Yaskawa INFORM job: SKRZYNIA_4640_-90_STOPNI_10BR.JBI

/JOB
//NAME SKRZYNIA_4640_-90_STOPNI_10BR
///FOLDERNAME 02-SKRZYNIE_JOBS
//POS
///NPOS 666,666,0,47,0,0
///TOOL 0
///POSTYPE PULSE
///PULSE
C00000=0,-52280,40443,0,6876,0
C00001=-82314,-24956,17040,-59626,-27382,-6248
C00002=-93910,-8625,17040,-59626,-43355,-6248
C00003=-98846,-1061,-42166,-80308,-57081,16120
C00004=-100452,6057,-48127,-85711,-56704,21322
C00005=-96957,25597,-37888,-85158,-62082,25522
C00006=-95580,33075,-33256,-84644,-64024,26851
C00007=-94380,33739,-32188,-85134,-63496,26721
C00008=-95580,33075,-33256,-84644,-64024,26851
C00009=-94940,31262,-36138,-85248,-63712,27160
C00010=-95580,33075,-33256,-84644,-64024,26851
C00011=-95263,33142,-33256,-84677,-63995,26850
C00012=-95263,33142,-33256,-84677,-63995,26850
C00013=-94261,33702,-32359,-85087,-63552,26740
C00014=-95263,33142,-33256,-84677,-63995,26850
C00015=-94777,31773,-35433,-85135,-63758,27084
C00016=-95263,33142,-33256,-84677,-63995,26850
C00017=-95260,33144,-33256,-84678,-63995,26850
C00018=-95260,33144,-33256,-84678,-63995,26850
C00019=-94282,33689,-32380,-85076,-63563,26742
C00020=-95260,33144,-33256,-84678,-63995,26850
C00021=-94827,31920,-35204,-85086,-63784,27059
C00022=-95260,33144,-33256,-84678,-63995,26850
C00023=-95258,33145,-33257,-84676,-63996,26846
C00024=-95258,33145,-33257,-84676,-63996,26846
C00025=-94286,33686,-32387,-85074,-63568,26738
C00026=-95258,33145,-33257,-84676,-63996,26846
C00027=-94874,32057,-34990,-85039,-63809,27032
C00028=-95258,33145,-33257,-84676,-63996,26846
C00029=-95377,22848,-19980,-77610,-66139,18413
C00030=-95383,22536,-19091,-77284,-66299,17999
C00031=-94454,23123,-18267,-77513,-65785,17889
C00032=-95383,22536,-19091,-77284,-66299,17999
C00033=-94991,21279,-20843,-77511,-66022,18108
C00034=-95383,22536,-19091,-77284,-66299,17999
C00035=-95258,25631,32269,-66559,-75499,2416
C00036=-95258,25631,32269,-66559,-75499,2416
C00037=-94333,26371,33350,-66433,-74983,2224
C00038=-95258,25631,32269,-66559,-75499,2416
C00039=-94886,24142,30119,-66602,-75133,2534
C00040=-95258,25631,32269,-66559,-75499,2416
C00041=-99189,25294,31874,-88720,-76886,6359
C00042=-99241,29593,38161,-92696,-78880,6430
C00043=-98514,30143,38992,-92642,-78372,6377
C00044=-99241,29593,38161,-92696,-78880,6430
C00045=-98973,29806,38536,-92693,-79698,6341
C00046=-99241,29593,38161,-92696,-78880,6430
C00047=-97871,32974,47728,-100928,-77160,11375
C00048=-97482,34142,50625,-102456,-76680,12291
C00049=-96768,34808,51684,-102358,-76154,12246
C00050=-97504,36083,53738,-102448,-77517,11844
C00051=-97263,35860,53475,-102452,-77986,11780
C00052=-97504,36083,53738,-102448,-77517,11844
C00053=-100410,-1172,-854,-105537,-63273,18802
C00054=-79271,-37169,-30482,-103288,-47510,17696
C00055=-79271,-9415,41877,-76443,-46100,-604
C00056=-100699,17246,57649,-91568,-58011,5122
C00057=-100093,19087,27862,-95634,-72730,8691
C00058=-99472,28508,32136,-95947,-79676,10682
C00059=-98577,29153,33099,-95929,-79046,10644
C00060=-99472,28508,32136,-95947,-79676,10682
C00061=-99113,26771,29576,-96019,-79505,10911
C00062=-99472,28508,32136,-95947,-79676,10682
C00063=-99199,18818,35660,-68259,-73735,6208
C00064=-95720,15423,18785,-70454,-68603,10022
C00065=-95720,15423,18785,-70454,-68603,10022
C00066=-97322,30100,38585,-71742,-79662,10416
C00067=-96349,30901,39804,-71630,-79090,10224
C00068=-97322,30100,38585,-71742,-79662,10416
C00069=-97054,28837,36680,-71776,-79387,10556
C00070=-97322,30100,38585,-71742,-79662,10416
C00071=-97373,30352,38967,-71736,-79717,10385
C00072=-97373,30352,38967,-71736,-79717,10385
C00073=-96432,31128,40151,-71627,-79165,10198
C00074=-97373,30352,38967,-71736,-79717,10385
C00075=-97071,28917,36802,-71776,-79407,10544
C00076=-97373,30352,38967,-71736,-79717,10385
C00077=-97356,30262,38827,-71739,-79698,10398
C00078=-97356,30262,38827,-71739,-79698,10398
C00079=-96507,30957,39891,-71642,-79201,10230
C00080=-97356,30262,38827,-71739,-79698,10398
C00081=-97092,29010,36937,-71773,-79425,10538
C00082=-97356,30262,38827,-71739,-79698,10398
C00083=-99745,23507,8579,-87147,-79275,20063
C00084=-99745,23568,9251,-87081,-79277,19867
C00085=-98882,24102,10002,-87178,-78701,19809
C00086=-99745,23568,9251,-87081,-79277,19867
C00087=-99406,22118,7226,-87176,-79050,20009
C00088=-99745,23568,9251,-87081,-79277,19867
C00089=-99071,22682,8038,-99994,-80807,17980
C00090=-99209,25375,15159,-99348,-81562,16520
C00091=-98424,25891,15901,-99427,-81018,16519
C00092=-99209,25375,15159,-99348,-81562,16520
C00093=-98879,23940,13118,-99425,-81414,16690
C00094=-99209,25375,15159,-99348,-81562,16520
C00095=-97630,34865,50283,-105962,-77348,9129
C00096=-97167,37263,56205,-105494,-76312,8157
C00097=-96392,38071,57532,-105366,-75722,8098
C00098=-97167,37263,56205,-105494,-76312,8157
C00099=-96830,35301,53019,-105613,-76328,8514
C00100=-97167,37263,56205,-105494,-76312,8157
C00101=-98819,19954,1043,-111479,-83154,14713
C00102=-100194,5325,-45038,-118611,-84970,27548
C00103=-77958,-36127,-88985,-138175,-66584,26591
C00104=-62749,-65297,-81682,-146767,-31843,20298
C00105=-53629,-59560,-53714,-89083,-24254,-4356
C00106=-73187,-23116,26488,-26118,-57509,-28469
C00107=-96139,-22548,-25766,-67560,-51232,-5154
C00108=-98398,-8109,-25057,-81551,-55130,4513
C00109=-99451,17861,2757,-80571,-73406,6045
C00110=-99056,24650,11359,-80216,-77425,5946
C00111=-98115,25261,12228,-80295,-76818,5843
C00112=-99056,24650,11359,-80216,-77425,5946
C00113=-98800,23560,9817,-80291,-77224,6050
C00114=-99056,24650,11359,-80216,-77425,5946
C00115=-99819,33446,48735,-87787,-79679,-1235
C00116=-99819,33446,48735,-87787,-79679,-1235
C00117=-98945,34179,49898,-87659,-79086,-1350
C00118=-99819,33446,48735,-87787,-79679,-1235
C00119=-99591,32133,46677,-87830,-79529,-1033
C00120=-99819,33446,48735,-87787,-79679,-1235
C00121=-98841,-14263,-23955,-101504,-55644,8170
C00122=-96175,-21848,-39130,-108881,-63715,10829
C00123=-56537,-51855,-41447,-79827,-26849,-3300
C00124=-37962,-64638,6899,-31784,1461,6885
C00125=0,-43112,23163,32261,-40956,29092
C00126=-38075,-37396,2384,-17964,-21120,46852
C00127=-50509,-19000,10610,-51503,-15997,61182
C00128=-53130,-17211,12007,-56251,-17152,63186
C00129=-51822,-15992,12994,-55136,-16324,62798
C00130=-53635,-15431,13457,-57815,-17251,63894
C00131=-53130,-17211,12007,-56251,-17152,63186
C00132=-50704,-18403,11069,-52157,-16018,61478
C00133=-53231,-16470,14622,-53206,-17893,61673
C00134=-51756,-15101,15744,-51790,-16990,61165
C00135=-53741,-14453,16285,-54808,-17949,62397
C00136=-53231,-17580,11714,-56182,-17246,63139
C00137=-51814,-19410,10295,-53186,-16720,61844
C00138=-53629,-18979,7405,-62018,-16535,65958
C00139=-52238,-17698,8415,-61175,-15613,65699
C00140=-53551,-17401,8655,-62910,-16346,66402
C00141=-52880,-17654,11656,-55678,-17066,62935
C00142=-51005,-17995,11387,-52847,-16122,61778
C00143=-52964,-17611,11689,-55811,-17106,62990
C00144=-51611,-16353,12697,-54642,-16249,62582
C00145=-53495,-15765,13180,-57466,-17201,63739
C00146=-52964,-17611,11689,-55811,-17106,62990
C00147=-51030,-17982,11395,-52891,-16135,61798
C00148=-52975,-17563,11726,-55850,-17109,63009
C00149=-51607,-16289,12749,-54669,-16241,62596
C00150=-53283,-15811,13140,-57177,-17094,63622
C00151=-52975,-17563,11726,-55850,-17109,63009
C00152=-50945,-18019,11363,-52741,-16103,61737
C00153=-52728,-17788,11545,-55393,-17010,62816
C00154=-51045,-16207,12813,-53894,-15944,62287
C00155=-52895,-15647,13274,-56746,-16874,63461
C00156=-52728,-17788,11545,-55393,-17010,62816
C00157=-50945,-18019,11363,-52741,-16103,61737
C00158=-52556,-17520,11756,-55311,-16888,62798
C00159=-51113,-16157,12849,-54025,-15975,62343
C00160=-52730,-15718,13210,-56498,-16792,63358
C00161=-52556,-17520,11756,-55311,-16888,62798
C00162=-50945,-18019,11363,-52741,-16103,61737
C00163=-51893,-17787,11546,-54246,-16568,62356
C00164=-50379,-16341,12703,-52826,-15610,61849
C00165=-52406,-15704,13225,-56071,-16614,63190
C00166=-51893,-17787,11546,-54246,-16568,62356
C00167=-50028,-22953,-3957,-22347,-31919,54220
C00168=-50947,-22502,-3625,-23433,-32061,54736
C00169=-49421,-20951,-2455,-21951,-31329,54057
C00170=-51207,-20433,-2055,-24026,-31698,55041
C00171=-50529,-22709,-3778,-22940,-31995,54502
C00172=-49763,-25421,-36239,-24565,-26935,60445
C00173=-49763,-25421,-36239,-24565,-26935,60445
C00174=-48299,-23485,-34758,-23276,-26122,59713
C00175=-50218,-22723,-34165,-25568,-26529,60993
C00176=-49763,-25421,-36239,-24565,-26935,60445
C00177=-50713,-12366,-58367,-41124,-17813,74400
C00178=-50824,-12254,-58263,-41255,-17847,74484
C00179=-49431,-10052,-56192,-40383,-17131,73813
C00180=-50915,-9358,-55524,-41955,-17664,74847
C00181=-51028,-12852,-58814,-41301,-17980,74542
C00182=-49763,-25421,-36239,-24565,-26935,60445
C00183=-50529,-22709,-3778,-22940,-31995,54502
C00184=-45389,-28224,4312,-35967,-15579,54278
C00185=-40154,-51179,-915,-24203,-8234,36524
C00186=0,-52280,40443,0,6876,0
C00187=0,-52280,40443,0,6876,0
C00188=-2117,-50103,-33543,-4117,45077,85249
C00189=26439,-48928,-33543,-4117,-52362,85249
C00190=26439,-27355,-33543,-41485,-52362,85249
C00191=39218,-24492,-41653,-51934,-39374,86964
C00192=39218,-24492,-41653,-51934,-39374,86964
C00193=46639,7575,-9331,-26045,-41627,82486
C00194=47278,8641,-9483,-26175,-40625,82510
C00195=46369,10567,-7126,-26545,-41054,82831
C00196=47278,8641,-9483,-26175,-40625,82510
C00197=48256,9506,-8430,-25641,-40400,82076
C00198=47278,8641,-9483,-26175,-40625,82510
C00199=44522,-635,-31983,-49264,-28311,89687
C00200=44247,-628,-31975,-49394,-28443,89790
C00201=43310,1314,-29842,-49807,-28910,90140
C00202=44247,-628,-31975,-49394,-28443,89790
C00203=45313,152,-31124,-48894,-27920,89380
C00204=44247,-628,-31975,-49394,-28443,89790
C00205=41572,-13073,-22520,-50760,-38355,84033
C00206=21909,-6773,-14577,-94161,-56302,89381
C00207=23773,-3183,-10897,-94486,-55065,89563
C00208=24904,-823,-8382,-94654,-54308,89644
C00209=24395,1151,-6219,-94590,-54651,89617
C00210=24904,-823,-8382,-94654,-54308,89644
C00211=26178,-337,-7854,-94816,-53451,89710
C00212=24904,-823,-8382,-94654,-54308,89644
C00213=17020,-16061,-23281,-93084,-59494,88637
C00214=-21568,-26506,-31664,-90508,-85573,86639
C00215=-8557,-39769,-22319,-51419,-69406,84680
C00216=-8557,-39769,-22319,-51419,-69406,84680
C00217=32994,-9735,-10751,-29019,-59471,69498
C00218=43974,9628,-22604,-36190,-36396,73426
C00219=45932,13115,-22315,-37472,-33732,73846
C00220=45228,14664,-20329,-37571,-34159,74020
C00221=45932,13115,-22315,-37472,-33732,73846
C00222=46653,13731,-21526,-37109,-33514,73520
C00223=45932,13115,-22315,-37472,-33732,73846
C00224=39039,866,-6986,-42761,-44691,67687
C00225=30717,-9248,-22721,-77433,-42696,79486
C00226=32434,-7077,-20587,-77571,-41526,79457
C00227=31883,-5576,-19073,-77676,-41878,79560
C00228=32434,-7077,-20587,-77571,-41526,79457
C00229=33092,-6769,-20280,-77576,-41084,79417
C00230=32434,-7077,-20587,-77571,-41526,79457
C00231=30527,-14106,-27266,-76898,-42917,79150
C00232=25454,-9581,-17335,-94425,-53880,89429
C00233=24965,-2445,-10120,-94645,-54263,89631
C00234=24893,-1278,-8874,-94650,-54314,89639
C00235=24417,557,-6877,-94595,-54636,89618
C00236=24893,-1278,-8874,-94650,-54314,89639
C00237=25752,-956,-8526,-94759,-53737,89684
C00238=24893,-1278,-8874,-94650,-54314,89639
C00239=23817,-1527,-9142,-94518,-55040,89587
C00240=24871,-1152,-8735,-94651,-54328,89643
C00241=24440,508,-6926,-94601,-54619,89624
C00242=24871,-1152,-8735,-94651,-54328,89643
C00243=25635,-865,-8427,-94748,-53815,89684
C00244=24871,-1152,-8735,-94651,-54328,89643
C00245=33203,-4295,-13750,-123758,-49995,81034
C00246=35028,4195,-6818,-132965,-58836,87950
C00247=35028,4195,-6818,-132965,-58836,87950
C00248=34452,5837,-4911,-132720,-59045,87770
C00249=35028,4195,-6818,-132965,-58836,87950
C00250=35710,4593,-6360,-133217,-58512,88125
C00251=35028,4195,-6818,-132965,-58836,87950
C00252=24762,-11408,-28656,-113055,-60293,85383
C00253=-28645,-26349,-41223,-103369,-91870,78302
C00254=-28645,-26349,-41223,-103369,-91870,78302
C00255=-25549,-24286,-26215,-66769,-87032,80148
C00256=27561,-8271,-12315,-63268,-52553,74387
C00257=29336,-165,-3925,-63163,-51316,74265
C00258=29518,765,-2904,-63127,-51205,74233
C00259=28850,2962,-447,-63227,-51636,74327
C00260=29518,765,-2904,-63127,-51205,74233
C00261=30662,1292,-2320,-62902,-50501,74035
C00262=29518,765,-2904,-63127,-51205,74233
C00263=30773,10953,32136,-106912,-46141,83783
C00264=30773,10953,32136,-106912,-46141,83783
C00265=30080,13410,35293,-106601,-46463,83481
C00266=30773,10953,32136,-106912,-46141,83783
C00267=32007,11622,32987,-106899,-45346,83915
C00268=30773,10953,32136,-106912,-46141,83783
C00269=28321,-8642,-16372,-95739,-47180,89965
C00270=28583,-7344,-15096,-95864,-47019,90043
C00271=27897,-5229,-12965,-95873,-47499,90079
C00272=28583,-7344,-15096,-95864,-47019,90043
C00273=29900,-6813,-14567,-96101,-46141,90154
C00274=28583,-7344,-15096,-95864,-47019,90043
C00275=27852,-7537,-15286,-95742,-47508,89986
C00276=28448,-7306,-15058,-95845,-47110,90035
C00277=27795,-5283,-13021,-95851,-47567,90065
C00278=28448,-7306,-15058,-95845,-47110,90035
C00279=29772,-6774,-14527,-96083,-46226,90146
C00280=28448,-7306,-15058,-95845,-47110,90035
C00281=18552,-19531,-26179,-93438,-53589,88597
C00282=40301,-14999,-52277,-148979,-69262,86714
C00283=42323,-33,-37432,-150113,-69667,87489
C00284=53245,19091,3515,-165691,-72595,90030
C00285=53641,19552,4138,-165817,-72473,90151
C00286=53058,20743,5761,-165615,-72317,89948
C00287=53641,19552,4138,-165817,-72473,90151
C00288=54155,20160,4967,-165982,-72308,90306
C00289=53641,19552,4138,-165817,-72473,90151
C00290=23439,-10154,-17205,-109204,-58547,76547
C00291=2382,-21913,-40813,-107544,-74451,77239
C00292=-31257,-15877,-35733,-102288,-96107,74463
C00293=-39204,-18003,-7668,-86141,-99190,68413
C00294=-5592,-5690,18047,-75373,-79525,63129
C00295=19039,-439,25862,-68224,-64120,61443
C00296=21624,5223,26011,-69375,-61155,63193
C00297=24437,11840,34139,-68260,-59598,62567
C00298=24053,13588,36402,-68249,-59917,62491
C00299=24437,11840,34139,-68260,-59598,62567
C00300=25079,12112,34488,-68051,-59212,62472
C00301=24437,11840,34139,-68260,-59598,62567
C00302=21370,4935,25667,-69451,-61310,63230
C00303=-18351,-11002,3811,-80352,-86206,66275
C00304=-34619,-5846,8788,-82342,-97004,67025
C00305=-40684,-19963,-8478,-86482,-100204,67987
C00306=1570,-13136,-5998,-86227,-71173,69099
C00307=13966,-6596,-2340,-86587,-62612,70052
C00308=24093,-1862,-9504,-94546,-54850,89594
C00309=24093,-1862,-9504,-94546,-54850,89594
C00310=23519,425,-7024,-94488,-55240,89573
C00311=24093,-1862,-9504,-94546,-54850,89594
C00312=25256,-1442,-9053,-94693,-54067,89656
C00313=24093,-1862,-9504,-94546,-54850,89594
C00314=27718,4364,12871,-105518,-51077,86669
C00315=27718,4364,12871,-105518,-51077,86669
C00316=27164,6353,15202,-105385,-51398,86539
C00317=27718,4364,12871,-105518,-51077,86669
C00318=28828,4851,13441,-105618,-50355,86801
C00319=27718,4364,12871,-105518,-51077,86669
C00320=20930,-1364,27707,-95004,-52134,77785
C00321=-41463,-32191,18163,-91991,-64949,55938
C00322=0,-52277,40442,0,6872,4
C00323=-82314,-24956,17040,-59626,-27382,-6248
C00324=-93910,-8625,17040,-59626,-43355,-6248
C00325=-98846,-1061,-42166,-80308,-57081,16120
C00326=-100452,6057,-48127,-85711,-56704,21322
C00327=-95564,34698,-34234,-85516,-63941,27819
C00328=-94221,34299,-28769,-82558,-65564,25844
C00329=-94107,37241,-30442,-84005,-65307,27544
C00330=-95103,32620,-31323,-83378,-64939,26072
C00331=-95103,32620,-31323,-83378,-64939,26072
C00332=-93990,32828,-31380,-83932,-64473,26160
C00333=-94063,31710,-30585,-83283,-64598,25457
C00334=-96692,32939,-31211,-82617,-65723,26190
C00335=-96111,21840,170,-71736,-70232,11396
C00336=-94229,22391,773,-71789,-70557,11468
C00337=-94283,22521,1025,-71678,-70686,11433
C00338=-95675,19167,-4176,-72970,-68231,11735
C00339=-95681,24338,3488,-71459,-71669,11415
C00340=-94245,22750,1246,-71757,-70674,11453
C00341=-94341,22923,1499,-71729,-70746,11440
C00342=-96213,24222,3324,-71394,-71999,11479
C00343=-95517,23330,2066,-71543,-71508,11507
C00344=-94304,22892,1449,-71738,-70721,11443
C00345=-94158,22889,1452,-71756,-70627,11429
C00346=-96071,24319,3461,-71408,-71916,11455
C00347=-96941,-6406,-33809,-76117,-54125,10511
C00348=-90643,-26862,-25633,-62597,-56791,-1368
C00349=-66103,-61757,7450,-21008,-32955,-5749
C00350=4223,-52290,40457,-5766,6913,3980
C00351=4223,-52290,40457,-5766,6913,3980
C00352=-4538,-50065,-33535,-3011,44998,84219
C00353=24207,-49248,-33668,-5551,-52644,86091
C00354=25094,-27722,-33812,-41887,-53054,85599
C00355=38036,-25052,-42086,-52219,-40087,87228
C00356=37328,-2824,-24733,-57182,-37821,90318
C00357=36700,-2520,-13735,-51589,-42201,86442
C00358=37520,2330,-3498,-48550,-43875,84431
C00359=37520,1020,-12079,-52650,-40851,87066
C00360=48458,-261,-12985,-24069,-43340,80504
C00361=36153,7296,-1758,-40139,-50302,89334
C00362=37146,11264,2520,-40849,-50296,89553
C00363=38059,11410,-1863,-40565,-47910,90206
C00364=36726,6476,-7858,-41213,-48206,90783
C00365=19339,7883,9818,-77509,-64249,74140
C00366=19027,1888,-16187,-103553,-67480,82955
C00367=24158,3537,-14322,-106039,-60939,84018
C00368=24143,4321,-7309,-103852,-59670,81875
C00369=19531,2904,-8928,-102027,-65985,80961
C00370=20232,-3383,-14682,-86495,-63009,78978
C00371=-24375,-51634,-49601,-83793,-94064,73950
C00372=4223,-52290,40457,-5766,6913,3980
C00373=-4825,-36686,24602,37792,-30278,35378
C00374=-46221,-29633,7403,-27051,-24124,46751
C00375=-46221,-29633,7403,-27051,-24124,46751
C00376=-52474,-20611,11454,-41004,-23045,52959
C00377=-60257,-19980,-2088,-84190,-23320,82051
C00378=-63868,-19883,-6318,-95759,-28031,88346
C00379=-51819,-22965,8574,-41365,-22900,53139
C00380=-4825,-36686,24602,37792,-30278,35378
C00381=0,-52280,40443,0,6876,0
C00382=4223,-52290,40457,-5766,6913,3980
C00383=-66103,-61757,7450,-21008,-32955,-5749
C00384=-89093,-33107,-44597,-67545,-52550,2722
C00385=-96941,-6406,-33809,-76117,-54125,10511
C00386=-99429,14378,84,-80785,-71596,8628
C00387=-99699,24313,24829,-82602,-77917,4569
C00388=-98066,26841,20697,-83331,-79245,6860
C00389=-98079,26929,20513,-83349,-79351,6953
C00390=-99638,19663,10292,-84193,-74452,7551
C00391=-98909,20891,5205,-92499,-77779,3679
C00392=-97991,21897,3469,-96150,-79490,1870
C00393=-97094,22407,2872,-101449,-80737,3094
C00394=-98052,22735,7381,-100906,-80646,1724
C00395=-96016,28471,32512,-109475,-77029,-270
C00396=-93697,27731,31018,-109675,-75757,229
C00397=-93697,30712,42128,-108463,-73689,-2160
C00398=-100174,9543,-9646,-113455,-77250,7387
C00399=-100174,1289,-12558,-103866,-68626,6781
C00400=-100177,-4656,-30138,-114506,-71921,12431
C00401=-97546,-19067,-24950,-97028,-60115,5718
C00402=-61441,-38616,11032,-55510,-42874,-3049
C00403=4223,-52290,40457,-5766,6913,3980
C00404=-22331,-23394,-30093,-82917,-82006,85712
C00405=22434,-14401,-3235,-51104,-60845,74728
C00406=42744,21307,45077,-24753,-69813,65333
C00407=33655,14083,18147,-45417,-58301,71861
C00408=33641,11943,8279,-47835,-54840,73983
C00409=36574,13250,23432,-35354,-61822,69159
C00410=28497,326,20939,-70981,-47632,72427
C00411=30972,5983,29862,-68494,-46670,70994
C00412=31029,11571,45127,-63398,-49004,67378
C00413=28971,8096,39948,-65070,-49810,68216
C00414=29759,-12862,-24221,-91747,-41905,86600
C00415=35278,-10419,-21940,-93284,-36771,87139
C00416=36208,-10883,-22374,-93618,-35345,87231
C00417=27219,-23595,-33313,-89555,-43517,85303
C00418=10564,-40773,-45889,-85382,-54876,82708
C00419=-14984,-61618,-24572,-87392,-53367,60735
C00420=9346,-67436,-18786,-75708,-34590,53709
C00421=40938,-55232,35946,-9746,5421,6718
C00422=4223,-52290,40457,-5766,6913,3980
C00423=-4825,-36686,24602,37792,-30278,35378
C00424=-46221,-29633,7403,-27051,-24124,46751
C00425=-56796,-22932,368,-68953,-21567,70907
C00426=-61611,-20349,-6598,-95791,-25091,88405
C00427=-62244,-19942,-5791,-95984,-25882,88372
C00428=-57752,-2938,32150,-100764,-20307,82364
C00429=-58257,-11045,22458,-94361,-23082,79795
C00430=-49294,-34086,9663,-30689,-30758,52546
C00431=4223,-52290,40457,-5766,6913,3980
C00432=0,-52280,40443,0,6876,0
C00433=0,-52280,40443,0,6876,0
C00434=-61754,-61602,7279,-16215,-32140,-7126
C00435=-89313,-24027,20291,-53466,-58905,-4975
C00436=-97807,-25409,-21837,-78881,-62828,2121
C00437=-100103,-15040,-13507,-79140,-58253,2724
C00438=-99725,9645,23361,-67154,-68568,-2059
C00439=-99271,16305,34765,-72797,-70067,-2351
C00440=-98402,25140,29245,-92090,-76944,4625
C00441=-98402,28265,40696,-90956,-76523,2010
C00442=-98754,23130,28932,-98122,-73671,5428
C00443=-98112,-9349,-13739,-99107,-55531,8873
C00444=-87692,-34175,-39658,-96739,-43399,8225
C00445=-75165,-16680,32803,-38944,-52307,-27215
C00446=-75165,-16680,32803,-38944,-52307,-27215
C00447=-96391,11374,61850,-52875,-60261,-22353
C00448=-96391,-17993,-25254,-79577,-45337,-1997
C00449=-84714,-13514,-21320,-79690,-37366,-2300
C00450=-92093,-5454,-13554,-80916,-52292,-613
C00451=-99761,24721,23429,-79408,-77929,-316
C00452=-99564,24916,23930,-79374,-77823,-417
C00453=-100005,27069,23687,-81767,-79755,895
C00454=-97295,30454,38512,-73622,-79542,-3831
C00455=-98471,27958,25022,-81751,-79627,782
C00456=-99805,23386,18402,-82055,-77455,1200
C00457=-100093,24719,20298,-81968,-77939,1081
C00458=-98451,26404,20171,-83400,-79044,-389
C00459=-98528,26732,19657,-84000,-79459,-654
C00460=-100109,23919,19160,-82044,-77303,1139
C00461=-98037,-4340,-16930,-86109,-58746,2389
C00462=-93345,-31758,-40240,-83703,-37467,-946
C00463=-81087,-35886,-14825,-53529,-36311,-18004
C00464=-47029,-49867,-20464,-11808,-29290,-36568
C00465=-41431,-67449,10869,-1325,127,-6150
C00466=6328,-52297,40483,-8599,6957,5944
C00467=-8648,-69005,-18270,-84275,-43232,53472
C00468=18757,-59462,-34892,-84638,-37529,67311
C00469=26772,-23733,-33422,-89486,-43820,85275
C00470=29039,-10071,-21608,-91386,-45181,86629
C00471=29639,-5923,-17523,-91591,-45648,86808
C00472=29709,-5453,-17046,-91618,-45636,86826
C00473=29138,-10182,-21714,-91372,-45196,86624
C00474=20424,-22725,-32635,-88800,-51006,85261
C00475=28416,-11420,-25238,-98178,-46636,84572
C00476=30481,-6584,-16425,-92636,-44382,82541
C00477=30464,-7521,-23523,-96665,-44944,85234
C00478=28416,-11420,-25238,-98178,-46636,84572
C00479=-23524,-33387,-42654,-89891,-81168,80229
C00480=-23524,-33387,-42654,-89891,-81168,80229
C00481=33935,-6399,-10013,-60506,-43064,77980
C00482=34878,-3211,-6740,-60356,-42422,77865
C00483=34873,-3218,-6748,-60357,-42424,77868
C00484=33935,-6399,-10013,-60506,-43064,77980
C00485=17782,-19597,1250,-60925,-51448,69151
C00486=-243,-43047,-13224,-69794,-55957,65877
C00487=42700,-55269,36176,-13619,5333,9062
C00488=6328,-52297,40483,-8599,6957,5944
C00489=-10231,-60460,6271,71658,-11927,-13637
C00490=-49129,-39322,3023,-34904,-18609,43900
C00491=-57258,-19535,13114,-46502,-25798,55150
C00492=-58736,-19151,1344,-78268,-22199,76919
C00493=-56868,-17231,8572,-62431,-21728,66645
C00494=-56011,-29317,6725,-41009,-27363,52457
C00495=-10137,-60963,4526,62308,-14518,-6745
C00496=0,-52280,40443,0,6876,0
C00497=0,-52280,40443,0,6876,0
C00498=-41653,-63035,2931,-3578,-7576,-14589
C00499=-45770,-50109,-20524,-10089,-29273,-37310
C00500=-80544,-36303,-15042,-52975,-36116,-18265
C00501=-93028,-32302,-40599,-83495,-37263,-1079
C00502=-98446,-3141,-15678,-86094,-59021,2414
C00503=-99951,24070,19376,-82000,-77829,1145
C00504=-98655,27908,24922,-81730,-79774,792
C00505=-98593,28720,26118,-81685,-80145,709
C00506=-99951,24070,19376,-82000,-77829,1145
C00507=-99951,24070,19376,-82000,-77829,1145
C00508=-98577,27118,23759,-81796,-79157,859
C00509=-98518,28577,26461,-81649,-79882,537
C00510=-99951,24070,19376,-82000,-77829,1145
C00511=-100023,27130,33022,-92975,-78123,-161
C00512=-98580,26185,31637,-93003,-77167,-1
C00513=-98580,30404,46303,-91600,-76541,-3267
C00514=-100724,18056,24349,-92081,-73134,-455
C00515=-98404,-4962,-6255,-93190,-58383,1895
C00516=-99487,-12045,-28221,-93829,-57357,5545
C00517=-95086,-30272,-46998,-91958,-53375,4609
C00518=-81694,-37220,-20464,-64791,-45723,-12569
C00519=-45770,-50109,-20524,-10089,-29273,-37310
C00520=-40984,-65135,6743,-2520,-4051,-10897
C00521=0,-52280,40443,0,6876,0
C00522=40939,-55232,35946,-9746,5421,6719
C00523=8707,-69002,-18268,-75213,-34271,52581
C00524=23267,-58917,-25142,-81990,-31707,62852
C00525=27307,-5613,10331,-81857,-46454,76095
C00526=30064,-5598,-963,-91827,-44222,81590
C00527=30419,-1725,5291,-88668,-43977,80354
C00528=30554,-300,10432,-88528,-43656,79164
C00529=29815,-6351,-3652,-90193,-44535,81892
C00530=29567,1847,27834,-65726,-48411,69959
C00531=23257,11670,30420,-81328,-57342,77033
C00532=23257,16856,45442,-77525,-58254,73578
C00533=21577,7912,33836,-78698,-59121,74340
C00534=17856,-9033,24892,-70658,-55966,67475
C00535=20838,-7097,2019,-111788,-62648,79114
C00536=40635,280,-7982,-142398,-56681,90238
C00537=32653,-9455,434,-90251,-40347,77213
C00538=40635,572,-6271,-142064,-55879,89947
C00539=40665,7761,2001,-141975,-55632,89869
C00540=40707,9678,10648,-140211,-51894,88431
C00541=39416,1907,3178,-139370,-51839,87774
C00542=7767,-21333,-19174,-120411,-69473,77116
C00543=33666,-18553,20064,-54519,-41956,59729
C00544=4032,-43511,13506,-33366,-30942,40837
C00545=22997,-56875,21315,16958,-8102,3163
C00546=0,-52280,40443,0,6876,0
C00547=-50974,-46557,23391,-77768,-13896,42026
C00548=-53474,-39983,4253,-39182,-18848,44272
C00549=-56619,-19856,12878,-45665,-25558,54806
C00550=-53298,-26712,-11188,-26889,-32979,52528
C00551=-57200,-20845,-7559,-37425,-33513,53351
C00552=-58648,-23818,-25853,-45100,-31207,62168
C00553=-58477,-22145,-38977,-48305,-29254,64725
C00554=-51868,-27423,-11673,-25269,-32728,51737
C00555=-49121,-45409,-2608,-26656,-19965,38583
C00556=-21301,-61008,4568,43957,-10534,-712
C00557=0,-52280,40443,0,6876,0
C00558=0,-52280,40443,0,6876,0
C00559=-40221,-67507,11044,-1325,-65,-6716
C00560=-45770,-50109,-20525,-10088,-29274,-37311
C00561=-80544,-36303,-15042,-52975,-36116,-18265
C00562=-93028,-32301,-40599,-83495,-37262,-1079
C00563=-97841,-4898,-17503,-86112,-58614,2374
C00564=-97574,22325,42435,-102650,-66613,-1893
C00565=-95754,35899,57018,-103970,-74003,-2798
C00566=-95754,43745,77672,-101743,-71699,-6650
C00567=-99714,17597,9613,-108150,-76803,6279
C00568=-93796,-17226,-33718,-118170,-55432,13587
C00569=-66816,-54797,-57006,-119089,-33370,13303
C00570=-66816,-52758,-50486,-115256,-31854,11154
C00571=-98141,-7636,2315,-105626,-50514,3722
C00572=-99521,20918,46679,-89083,-66665,-5358
C00573=-98691,34973,58126,-90608,-76643,-4580
C00574=-98691,42061,76615,-89053,-76304,-8086
C00575=-98720,15018,65588,-59406,-66947,-17238
C00576=-93628,-24224,-10838,-81898,-52333,-4131
C00577=-86170,-37737,-28198,-69261,-47898,-9342
C00578=-45770,-50109,-20525,-10088,-29274,-37311
C00579=-40221,-67507,11044,-1325,-65,-6716
C00580=0,-52280,40443,0,6876,0
C00581=51241,-30653,28678,4016,-29070,6398
C00582=46185,-61941,-37286,-12736,-10732,51851
C00583=-13205,-44768,-23966,-65315,-59418,73750
C00584=-11120,-40541,-20876,-69249,-61539,75403
C00585=-836,-13033,12361,-83908,-73576,73378
C00586=18912,6214,32354,-79489,-60743,73080
C00587=21217,10898,38129,-78632,-59343,72736
C00588=23447,16313,45262,-77527,-58074,72177
C00589=23610,23756,64158,-73325,-59549,68283
C00590=18912,6214,32354,-79489,-60743,73080
C00591=-836,-13033,12361,-83908,-73576,73378
C00592=-20209,-39682,-20467,-71924,-67122,76479
C00593=-20209,-39682,-20467,-71924,-67122,76479
C00594=26353,-3691,11741,-61723,-54035,71160
C00595=29598,-2090,11073,-69087,-47235,76987
C00596=30217,-1844,4641,-75777,-45517,79979
C00597=29529,1742,11379,-68166,-49318,73572
C00598=24010,-9039,-4437,-79986,-50972,77255
C00599=24652,-10740,-12845,-99298,-50700,81949
C00600=28976,-2672,-4778,-100308,-47937,82653
C00601=31030,-2921,-9996,-112394,-49006,86348
C00602=24652,-10740,-12845,-99298,-50700,81949
C00603=-25637,-26222,-38592,-96633,-85474,81576
C00604=-36771,-16470,-4689,-95304,-89579,74076
C00605=-33704,-12343,7746,-85568,-87064,70052
C00606=4032,-43511,13506,-33366,-30942,40837
C00607=27500,-60047,23168,28912,-2679,-5784
C00608=0,-52280,40443,0,6876,0
C00609=-50971,-46557,23390,-77766,-13895,42026
C00610=-53475,-39984,4253,-39182,-18848,44273
C00611=-56619,-19856,12878,-45665,-25558,54806
C00612=-57643,-27958,-8553,-51854,-24771,59787
C00613=-66195,-24410,-19095,-90567,-31132,85904
C00614=-63290,-24193,-14362,-80030,-27547,78073
C00615=-39040,-40975,-15408,-18643,-21575,44866
C00616=-11647,-69843,-10959,56399,-11165,-4616
C00617=-15394,-57237,30542,-10392,5525,8219
C00618=0,-52280,40443,0,6876,0
C00619=0,-52280,40443,0,6876,0
C00620=-40221,-67507,11044,-1325,-65,-6716
C00621=-45770,-50109,-20525,-10088,-29274,-37311
C00622=-95022,-19559,-3970,-66108,-42168,-11789
C00623=-84972,-7110,7117,-67721,-41324,-10731
C00624=-83869,-8155,6098,-67213,-40658,-10968
C00625=-99927,23961,20220,-85683,-78298,772
C00626=-98562,26853,28284,-85090,-78334,-823
C00627=-98562,24944,18750,-86001,-78172,1594
C00628=-99530,24174,17652,-85964,-78826,1685
C00629=-98491,25445,31196,-89357,-76395,-673
C00630=-98197,26014,32882,-93044,-76072,-339
C00631=-99839,23064,19027,-85806,-76881,822
C00632=-86774,-13232,-16630,-85484,-41019,-1154
C00633=-97999,-21060,-29835,-88214,-48653,956
C00634=-98846,-3268,25064,-74217,-51189,-12584
C00635=-70313,-35289,-4922,-51188,-38634,-20596
C00636=-81694,-37221,-20464,-64791,-45723,-12569
C00637=-45770,-50109,-20525,-10088,-29274,-37311
C00638=-41628,-63095,3038,-3547,-7472,-14475
C00639=4223,-52290,40457,-5766,6913,3980
C00640=4224,-52288,40457,-5773,6909,3978
C00641=4224,-52288,40457,-28770,-64753,45638
C00642=6548,2882,44080,-77825,-67624,70557
C00643=22702,21750,69443,-66118,-61597,67582
C00644=25585,21999,63350,-62249,-61285,68688
C00645=25777,17209,50811,-62979,-59886,70957
C00646=23226,22825,71113,-65575,-61542,67353
C00647=24931,14697,51677,-80718,-51653,72069
C00648=24746,14409,39758,-87518,-53542,76879
C00649=24784,21556,58944,-82031,-53873,72431
C00650=22657,12722,42993,-85587,-54940,74916
C00651=-4427,-20395,-7318,-104668,-69521,79317
C00652=768,-20151,-3587,-97758,-65802,76626
C00653=-14736,-21545,-1233,-93598,-60476,72578
C00654=1642,-46684,14475,-47609,-24983,34912
C00655=27500,-60047,23168,28912,-2679,-5784
C00656=0,-52280,40443,0,6876,0
C00657=-50971,-46557,23390,-77766,-13895,42026
C00658=-53475,-39984,4253,-39182,-18848,44273
C00659=-56619,-19856,12878,-45665,-25558,54806
C00660=-53891,-17708,14512,-43170,-23995,53902
C00661=-60674,-17500,6427,-71116,-24772,71097
C00662=-63181,-17997,2063,-82122,-26831,78394
C00663=-39402,-27697,7664,-17904,-21663,43170
C00664=-11647,-69843,-10959,56399,-11165,-4616
C00665=0,-52280,40443,0,6876,0
BC00000=464364
BC00001=445130
BC00002=445130
BC00003=445130
BC00004=445130
BC00005=445130
BC00006=445130
BC00007=445130
BC00008=445130
BC00009=445130
BC00010=445130
BC00011=491232
BC00012=491232
BC00013=491232
BC00014=491232
BC00015=491232
BC00016=491232
BC00017=537442
BC00018=537442
BC00019=537442
BC00020=537442
BC00021=537442
BC00022=537442
BC00023=583546
BC00024=583546
BC00025=583546
BC00026=583546
BC00027=583546
BC00028=583546
BC00029=573543
BC00030=573053
BC00031=573053
BC00032=573053
BC00033=573054
BC00034=573053
BC00035=559393
BC00036=559393
BC00037=559393
BC00038=559393
BC00039=559393
BC00040=559393
BC00041=556308
BC00042=555729
BC00043=555729
BC00044=555729
BC00045=555729
BC00046=555729
BC00047=559296
BC00048=560018
BC00049=560018
BC00050=560018
BC00051=560018
BC00052=560018
BC00053=523222
BC00054=523222
BC00055=570475
BC00056=604868
BC00057=615389
BC00058=626919
BC00059=626919
BC00060=626919
BC00061=626919
BC00062=626919
BC00063=714117
BC00064=714117
BC00065=714117
BC00066=714117
BC00067=714117
BC00068=714117
BC00069=714117
BC00070=714117
BC00071=737203
BC00072=737203
BC00073=737203
BC00074=737203
BC00075=737203
BC00076=737203
BC00077=783275
BC00078=783275
BC00079=783275
BC00080=783275
BC00081=783275
BC00082=783275
BC00083=806364
BC00084=806364
BC00085=806363
BC00086=806364
BC00087=806364
BC00088=806364
BC00089=813588
BC00090=813588
BC00091=813588
BC00092=813588
BC00093=813588
BC00094=813588
BC00095=798005
BC00096=798005
BC00097=798005
BC00098=798005
BC00099=798005
BC00100=798005
BC00101=798393
BC00102=807318
BC00103=833381
BC00104=907576
BC00105=902087
BC00106=891348
BC00107=924005
BC00108=930620
BC00109=930645
BC00110=930651
BC00111=930651
BC00112=930651
BC00113=930651
BC00114=930651
BC00115=911614
BC00116=926975
BC00117=926975
BC00118=926975
BC00119=926975
BC00120=926975
BC00121=927828
BC00122=917545
BC00123=909325
BC00124=773205
BC00125=811795
BC00126=896888
BC00127=889624
BC00128=889624
BC00129=889624
BC00130=889624
BC00131=889624
BC00132=828182
BC00133=828182
BC00134=828182
BC00135=828182
BC00136=828182
BC00137=766752
BC00138=766752
BC00139=766752
BC00140=766752
BC00141=766752
BC00142=705350
BC00143=705350
BC00144=705350
BC00145=705350
BC00146=705350
BC00147=643865
BC00148=643865
BC00149=643865
BC00150=643865
BC00151=643865
BC00152=582464
BC00153=582464
BC00154=582464
BC00155=582464
BC00156=582464
BC00157=520992
BC00158=520992
BC00159=520992
BC00160=520992
BC00161=520992
BC00162=459540
BC00163=459540
BC00164=459540
BC00165=459540
BC00166=459540
BC00167=459544
BC00168=459544
BC00169=459544
BC00170=459544
BC00171=459544
BC00172=459544
BC00173=459544
BC00174=459544
BC00175=459544
BC00176=459544
BC00177=459544
BC00178=459544
BC00179=459544
BC00180=459544
BC00181=459544
BC00182=459544
BC00183=459544
BC00184=459540
BC00185=533216
BC00186=533216
BC00187=492150
BC00188=423885
BC00189=423885
BC00190=423885
BC00191=423885
BC00192=423885
BC00193=493160
BC00194=493160
BC00195=493160
BC00196=493160
BC00197=493160
BC00198=493160
BC00199=539180
BC00200=539180
BC00201=539180
BC00202=539180
BC00203=539180
BC00204=539180
BC00205=525487
BC00206=485388
BC00207=485386
BC00208=485384
BC00209=485384
BC00210=485384
BC00211=485384
BC00212=485384
BC00213=485384
BC00214=485384
BC00215=485384
BC00216=635507
BC00217=635507
BC00218=635507
BC00219=635509
BC00220=635509
BC00221=635509
BC00222=635509
BC00223=635509
BC00224=603035
BC00225=594948
BC00226=594948
BC00227=594948
BC00228=594948
BC00229=594948
BC00230=594948
BC00231=594948
BC00232=600591
BC00233=600589
BC00234=600589
BC00235=600589
BC00236=600589
BC00237=600589
BC00238=600589
BC00239=623637
BC00240=623637
BC00241=623637
BC00242=623637
BC00243=623637
BC00244=623637
BC00245=623637
BC00246=623637
BC00247=623637
BC00248=623637
BC00249=623637
BC00250=623637
BC00251=623637
BC00252=623637
BC00253=623637
BC00254=758391
BC00255=758391
BC00256=758391
BC00257=758391
BC00258=758391
BC00259=758391
BC00260=758391
BC00261=758391
BC00262=758391
BC00263=669704
BC00264=669704
BC00265=669706
BC00266=669704
BC00267=669704
BC00268=669704
BC00269=784942
BC00270=784942
BC00271=784942
BC00272=784942
BC00273=784942
BC00274=784942
BC00275=807985
BC00276=807985
BC00277=807985
BC00278=807985
BC00279=807985
BC00280=807985
BC00281=807985
BC00282=784942
BC00283=784942
BC00284=784942
BC00285=784942
BC00286=784942
BC00287=784942
BC00288=784942
BC00289=784942
BC00290=785203
BC00291=785203
BC00292=785203
BC00293=895226
BC00294=895226
BC00295=895226
BC00296=895226
BC00297=895226
BC00298=895226
BC00299=895226
BC00300=895226
BC00301=895226
BC00302=895226
BC00303=906894
BC00304=906894
BC00305=963281
BC00306=963281
BC00307=963281
BC00308=969297
BC00309=969297
BC00310=969297
BC00311=969297
BC00312=969297
BC00313=969297
BC00314=969297
BC00315=969297
BC00316=969297
BC00317=969297
BC00318=969297
BC00319=969297
BC00320=927243
BC00321=883644
BC00322=475149
BC00323=445130
BC00324=445130
BC00325=445130
BC00326=445130
BC00327=445130
BC00328=445710
BC00329=445126
BC00330=445722
BC00331=484130
BC00332=492177
BC00333=481766
BC00334=492273
BC00335=473247
BC00336=480563
BC00337=473247
BC00338=480984
BC00339=519338
BC00340=527043
BC00341=519335
BC00342=519335
BC00343=550079
BC00344=550079
BC00345=542403
BC00346=542207
BC00347=506510
BC00348=542207
BC00349=519224
BC00350=542207
BC00351=492150
BC00352=423885
BC00353=471005
BC00354=487965
BC00355=477405
BC00356=472948
BC00357=455020
BC00358=453643
BC00359=453643
BC00360=493160
BC00361=521199
BC00362=521199
BC00363=521199
BC00364=521199
BC00365=484684
BC00366=484684
BC00367=484684
BC00368=484684
BC00369=484684
BC00370=484684
BC00371=484684
BC00372=493160
BC00373=582810
BC00374=655182
BC00375=655182
BC00376=655182
BC00377=655182
BC00378=716328
BC00379=716642
BC00380=582810
BC00381=493160
BC00382=542207
BC00383=542207
BC00384=505858
BC00385=590944
BC00386=557139
BC00387=543764
BC00388=551223
BC00389=543862
BC00390=551454
BC00391=569700
BC00392=577961
BC00393=577961
BC00394=577961
BC00395=553908
BC00396=553908
BC00397=553908
BC00398=553908
BC00399=556944
BC00400=553210
BC00401=547251
BC00402=533724
BC00403=584417
BC00404=590475
BC00405=610524
BC00406=594969
BC00407=594969
BC00408=594969
BC00409=593583
BC00410=552811
BC00411=552811
BC00412=552811
BC00413=552811
BC00414=612529
BC00415=612529
BC00416=620193
BC00417=620193
BC00418=620193
BC00419=620193
BC00420=620193
BC00421=620193
BC00422=620193
BC00423=812803
BC00424=887783
BC00425=897274
BC00426=900756
BC00427=919707
BC00428=882885
BC00429=879096
BC00430=853059
BC00431=542207
BC00432=542207
BC00433=542207
BC00434=542207
BC00435=601313
BC00436=638007
BC00437=633482
BC00438=625047
BC00439=623076
BC00440=621438
BC00441=621438
BC00442=621342
BC00443=625429
BC00444=630287
BC00445=633159
BC00446=681733
BC00447=681733
BC00448=740703
BC00449=740703
BC00450=740703
BC00451=740703
BC00452=710007
BC00453=710007
BC00454=703771
BC00455=710137
BC00456=710007
BC00457=727159
BC00458=725395
BC00459=733039
BC00460=733103
BC00461=733103
BC00462=733103
BC00463=733103
BC00464=733103
BC00465=733103
BC00466=733103
BC00467=620193
BC00468=626283
BC00469=635598
BC00470=635765
BC00471=635816
BC00472=643271
BC00473=641590
BC00474=641590
BC00475=685792
BC00476=685797
BC00477=685792
BC00478=685792
BC00479=685792
BC00480=771083
BC00481=750783
BC00482=758455
BC00483=750783
BC00484=750783
BC00485=719658
BC00486=685920
BC00487=620193
BC00488=620193
BC00489=561542
BC00490=498768
BC00491=407896
BC00492=407892
BC00493=469047
BC00494=469397
BC00495=524165
BC00496=524165
BC00497=733103
BC00498=733103
BC00499=733103
BC00500=733103
BC00501=733103
BC00502=733103
BC00503=771424
BC00504=771424
BC00505=779179
BC00506=771424
BC00507=794504
BC00508=794504
BC00509=801218
BC00510=794504
BC00511=789231
BC00512=789231
BC00513=789231
BC00514=791588
BC00515=794354
BC00516=814020
BC00517=820656
BC00518=840598
BC00519=795297
BC00520=741582
BC00521=733102
BC00522=620193
BC00523=700154
BC00524=704277
BC00525=716233
BC00526=716233
BC00527=716233
BC00528=716233
BC00529=716233
BC00530=733710
BC00531=733710
BC00532=733710
BC00533=733710
BC00534=742336
BC00535=742336
BC00536=742336
BC00537=763798
BC00538=742336
BC00539=742336
BC00540=742336
BC00541=742336
BC00542=743633
BC00543=750104
BC00544=672725
BC00545=672725
BC00546=672725
BC00547=576077
BC00548=465158
BC00549=407896
BC00550=407896
BC00551=407896
BC00552=407896
BC00553=407896
BC00554=407896
BC00555=471446
BC00556=524165
BC00557=524165
BC00558=733103
BC00559=733103
BC00560=733103
BC00561=733103
BC00562=733103
BC00563=733103
BC00564=782402
BC00565=790647
BC00566=790647
BC00567=792197
BC00568=792197
BC00569=792197
BC00570=850465
BC00571=850465
BC00572=847712
BC00573=860374
BC00574=860374
BC00575=860374
BC00576=842476
BC00577=853507
BC00578=795297
BC00579=733103
BC00580=733103
BC00581=762701
BC00582=816902
BC00583=816902
BC00584=837114
BC00585=816902
BC00586=816839
BC00587=816869
BC00588=816900
BC00589=816902
BC00590=816839
BC00591=816902
BC00592=837114
BC00593=903552
BC00594=903552
BC00595=897057
BC00596=903398
BC00597=903552
BC00598=903552
BC00599=903552
BC00600=903552
BC00601=903552
BC00602=903552
BC00603=903552
BC00604=848113
BC00605=815298
BC00606=672725
BC00607=672725
BC00608=672725
BC00609=576077
BC00610=513681
BC00611=534857
BC00612=557970
BC00613=557452
BC00614=618309
BC00615=618402
BC00616=618402
BC00617=618402
BC00618=618402
BC00619=733103
BC00620=733103
BC00621=915795
BC00622=908310
BC00623=908310
BC00624=908310
BC00625=931674
BC00626=931676
BC00627=931676
BC00628=931676
BC00629=931783
BC00630=931783
BC00631=932643
BC00632=928885
BC00633=920461
BC00634=899596
BC00635=883074
BC00636=840598
BC00637=795297
BC00638=748875
BC00639=733103
BC00640=852584
BC00641=921533
BC00642=921533
BC00643=923427
BC00644=923499
BC00645=923499
BC00646=923501
BC00647=932594
BC00648=943380
BC00649=943380
BC00650=943380
BC00651=963295
BC00652=934184
BC00653=929661
BC00654=754884
BC00655=672725
BC00656=672725
BC00657=749842
BC00658=756681
BC00659=776639
BC00660=776639
BC00661=776639
BC00662=838373
BC00663=837995
BC00664=796760
BC00665=742282
///POSTYPE BASE
///RECTAN
///RCONF 1,0,0,0,0,0,0,0,0,0,0,0,0,0,0,0,0,0,0,0,0,0,0,0
P00006=0.000,0.000,0.000,0.0000,0.0000,0.0000
///RCONF 0,0,0,0,0,0,0,0,0,0,0,0,0,0,0,0,0,0,0,0,0,0,0,0
P00058=0.000,0.000,3.000,0.0000,0.0000,0.0000
///RCONF 1,0,0,0,0,0,0,0,0,0,0,0,0,0,0,0,0,0,0,0,0,0,0,0
P00300=-0.036,-1.505,2.318,0.0000,0.0000,0.0000
P00301=0.046,-2.112,7.779,0.0000,0.0000,0.0000
P00302=-0.180,-2.409,6.326,0.0000,0.0000,0.0000
///RCONF 0,0,0,0,0,0,0,0,0,0,0,0,0,0,0,0,0,0,0,0,0,0,0,0
P00303=-0.004,-1.437,-4.584,0.0000,0.0000,0.0000
P00304=0.028,-1.666,-4.234,0.0000,0.0000,0.0000
P00305=-0.003,-1.920,-3.501,0.0000,0.0000,0.0000
P00306=0.015,-2.252,-3.054,0.0000,0.0000,0.0000
P00307=0.019,-2.151,-5.077,0.0000,0.0000,0.0000
P00308=-0.003,-2.092,-4.888,0.0000,0.0000,0.0000
P00309=-0.040,-2.205,-4.992,0.0000,0.0000,0.0000
P00310=-0.006,-2.490,-5.925,0.0000,0.0000,0.0000
P00311=-0.007,-2.079,-5.307,0.0000,0.0000,0.0000
P00312=-0.032,2.202,-7.632,0.0000,0.0000,0.0000
///RCONF 1,0,0,0,0,0,0,0,0,0,0,0,0,0,0,0,0,0,0,0,0,0,0,0
P00313=-0.088,1.055,2.110,0.0000,0.0000,0.0000
P00314=-0.055,1.752,1.634,0.0000,0.0000,0.0000
P00316=0.009,2.112,2.075,0.0000,0.0000,0.0000
P00317=-0.015,2.781,3.126,0.0000,0.0000,0.0000
///RCONF 0,0,0,0,0,0,0,0,0,0,0,0,0,0,0,0,0,0,0,0,0,0,0,0
P00351=13.563,-0.027,-0.653,0.0000,0.0000,0.0000
P00352=13.252,-0.027,-0.827,0.0000,0.0000,0.0000
P00353=10.971,-0.082,0.776,0.0000,0.0000,0.0000
P00354=-0.024,2.508,-1.824,0.0000,0.0000,0.0000
P00355=-0.001,2.528,-1.131,0.0000,0.0000,0.0000
P00356=-0.034,2.921,-0.262,0.0000,0.0000,0.0000
P00357=0.003,3.386,-0.091,0.0000,0.0000,0.0000
P00358=0.014,3.037,-0.020,0.0000,0.0000,0.0000
P00359=-0.005,2.731,0.912,0.0000,0.0000,0.0000
P00360=-0.011,3.412,0.438,0.0000,0.0000,0.0000
P00361=0.018,3.050,1.253,0.0000,0.0000,0.0000
P00401=3.430,-0.021,1.131,0.0000,0.0000,0.0000
P00402=-0.253,1.107,3.062,0.0000,0.0000,0.0000
P00403=-3.666,-0.015,5.328,0.0000,0.0000,0.0000
///RCONF 1,0,0,0,0,0,0,0,0,0,0,0,0,0,0,0,0,0,0,0,0,0,0,0
P00404=0.029,4.189,-1.030,0.0000,0.0000,0.0000
///RCONF 0,0,0,0,0,0,0,0,0,0,0,0,0,0,0,0,0,0,0,0,0,0,0,0
P00405=2.420,0.007,1.427,0.0000,0.0000,0.0000
P00406=3.513,-0.022,0.429,0.0000,0.0000,0.0000
///RCONF 1,0,0,0,1,0,0,0,0,0,0,0,0,0,0,0,0,0,0,0,0,0,0,0
P00407=-0.029,2.348,-1.469,0.0000,0.0000,0.0000
P00408=0.010,1.346,-1.479,0.0000,0.0000,0.0000
///RCONF 1,0,0,0,0,0,0,0,0,0,0,0,0,0,0,0,0,0,0,0,0,0,0,0
P00409=-0.026,2.090,-1.483,0.0000,0.0000,0.0000
P00410=0.001,4.491,-0.583,0.0000,0.0000,0.0000
///RCONF 1,0,0,0,1,0,0,0,0,0,0,0,0,0,0,0,0,0,0,0,0,0,0,0
P00411=-0.015,3.627,0.872,0.0000,0.0000,0.0000
P00412=0.002,3.829,0.787,0.0000,0.0000,0.0000
P00413=0.046,0.107,-0.040,0.0000,0.0000,0.0000
///RCONF 1,0,0,0,0,0,0,0,0,0,0,0,0,0,0,0,0,0,0,0,0,0,0,0
P00414=0.046,0.800,0.739,0.0000,0.0000,0.0000
///RCONF 0,0,0,0,0,0,0,0,0,0,0,0,0,0,0,0,0,0,0,0,0,0,0,0
P00415=-1.781,-1.303,3.250,0.0000,0.0000,0.0000
P00416=0.027,1.119,3.078,0.0000,0.0000,0.0000
///RCONF 1,0,0,0,1,0,0,0,0,0,0,0,0,0,0,0,0,0,0,0,0,0,0,0
P00417=0.059,4.721,3.973,0.0000,0.0000,0.0000
//INST
///DATE 2024/06/27 18:37
///ATTR SC,RW
///GROUP1 RB1,BS1
NOP
CALL JOB:MOVE_INTO_TUNNEL
MOVJ C00000 BC00000 VJ=50.00
MOVJ C00001 BC00001 VJ=40.00
MOVJ C00002 BC00002 VJ=40.00
MOVL C00003 BC00003 V=666.7
MOVJ C00004 BC00004 VJ=30.00
MOVL C00005 BC00005 V=500.0
'------------------------
'W31.2
'------------------------
MOVL C00006 BC00006 V=166.7 PL=0
REFP 3 C00007 BC00007
CALL JOB:SEARCH-R1
SET P0300 P0006
SFTON P0300
MOVL C00008 BC00008 V=166.7 PL=0
REFP 3 C00009 BC00009
CALL JOB:SEARCH-R1
SET P0300 P0006
SFTON P0300
MOVL C00010 BC00010 V=166.7 PL=0
SFTOF
'------------------------
'W31.4
'------------------------
MOVL C00011 BC00011 V=500.0
MOVL C00012 BC00012 V=166.7 PL=0
REFP 3 C00013 BC00013
CALL JOB:SEARCH-R1
SET P0301 P0006
SFTON P0301
MOVL C00014 BC00014 V=166.7 PL=0
REFP 3 C00015 BC00015
CALL JOB:SEARCH-R1
SET P0301 P0006
SFTON P0301
MOVL C00016 BC00016 V=166.7 PL=0
SFTOF
'------------------------
'W31.6
'------------------------
MOVL C00017 BC00017 V=500.0
MOVL C00018 BC00018 V=166.7 PL=0
REFP 3 C00019 BC00019
CALL JOB:SEARCH-R1
SET P0302 P0006
SFTON P0302
MOVL C00020 BC00020 V=166.7 PL=0
REFP 3 C00021 BC00021
CALL JOB:SEARCH-R1
SET P0302 P0006
SFTON P0302
MOVL C00022 BC00022 V=166.7 PL=0
SFTOF
'------------------------
'W31.8
'------------------------
MOVL C00023 BC00023 V=500.0
MOVL C00024 BC00024 V=166.7 PL=0
REFP 3 C00025 BC00025
CALL JOB:SEARCH-R1
SET P0303 P0006
SFTON P0303
MOVL C00026 BC00026 V=166.7 PL=0
REFP 3 C00027 BC00027
CALL JOB:SEARCH-R1
SET P0303 P0006
SFTON P0303
MOVL C00028 BC00028 V=166.7 PL=0
SFTOF
'------------------------
'W31.9
'------------------------
MOVL C00029 BC00029 V=500.0
MOVL C00030 BC00030 V=166.7 PL=0
REFP 3 C00031 BC00031
CALL JOB:SEARCH-R1
SET P0304 P0006
SFTON P0304
MOVL C00032 BC00032 V=166.7 PL=0
REFP 3 C00033 BC00033
CALL JOB:SEARCH-R1
SET P0304 P0006
SFTON P0304
MOVL C00034 BC00034 V=166.7 PL=0
SFTOF
'------------------------
'W31.11
'------------------------
MOVL C00035 BC00035 V=500.0
MOVL C00036 BC00036 V=166.7 PL=0
REFP 3 C00037 BC00037
CALL JOB:SEARCH-R1
SET P0305 P0006
SFTON P0305
MOVL C00038 BC00038 V=166.7 PL=0
REFP 3 C00039 BC00039
CALL JOB:SEARCH-R1
SET P0305 P0006
SFTON P0305
MOVL C00040 BC00040 V=166.7 PL=0
SFTOF
'------------------------
'W31.13
'------------------------
MOVL C00041 BC00041 V=500.0
MOVL C00042 BC00042 V=166.7 PL=0
REFP 3 C00043 BC00043
CALL JOB:SEARCH-R1
SET P0306 P0006
SFTON P0306
MOVL C00044 BC00044 V=166.7 PL=0
REFP 3 C00045 BC00045
CALL JOB:SEARCH-R1
SET P0306 P0006
SFTON P0306
MOVL C00046 BC00046 V=166.7 PL=0
SFTOF
'------------------------
'W31.14
'------------------------
MOVL C00047 BC00047 V=333.3
MOVL C00048 BC00048 V=166.7 PL=0
REFP 3 C00049 BC00049
CALL JOB:SEARCH-R1
SET P0307 P0006
SFTON P0307
MOVL C00050 BC00050 V=166.7 PL=0
REFP 3 C00051 BC00051
CALL JOB:SEARCH-R1
SET P0307 P0006
SFTON P0307
MOVL C00052 BC00052 V=166.7 PL=0
SFTOF
MOVL C00053 BC00053 V=500.0
MOVL C00054 BC00054 V=500.0
MOVL C00055 BC00055 V=500.0
MOVL C00056 BC00056 V=500.0
'------------------------
'W31.16
'------------------------
MOVL C00057 BC00057 V=500.0
MOVL C00058 BC00058 V=166.7 PL=0
REFP 3 C00059 BC00059
CALL JOB:SEARCH-R1
SET P0308 P0006
SFTON P0308
MOVL C00060 BC00060 V=166.7 PL=0
REFP 3 C00061 BC00061
CALL JOB:SEARCH-R1
SET P0308 P0006
SFTON P0308
MOVL C00062 BC00062 V=166.7 PL=0
SFTOF
MOVL C00063 BC00063 V=500.0
MOVL C00064 BC00064 V=333.3
'------------------------
'W31.18
'------------------------
MOVL C00065 BC00065 V=166.7
MOVL C00066 BC00066 V=133.3 PL=0
REFP 3 C00067 BC00067
CALL JOB:SEARCH-R1
SET P0309 P0006
SFTON P0309
MOVL C00068 BC00068 V=66.7 PL=0
REFP 3 C00069 BC00069
CALL JOB:SEARCH-R1
SET P0309 P0006
SFTON P0309
MOVL C00070 BC00070 V=66.7 PL=0
SFTOF
'------------------------
'W31.19
'------------------------
MOVL C00071 BC00071 V=500.0
MOVL C00072 BC00072 V=166.7 PL=0
REFP 3 C00073 BC00073
CALL JOB:SEARCH-R1
SET P0310 P0006
SFTON P0310
MOVL C00074 BC00074 V=166.7 PL=0
REFP 3 C00075 BC00075
CALL JOB:SEARCH-R1
SET P0310 P0006
SFTON P0310
MOVL C00076 BC00076 V=166.7 PL=0
SFTOF
'------------------------
'W31.21
'------------------------
MOVL C00077 BC00077 V=500.0
MOVL C00078 BC00078 V=166.7 PL=0
REFP 3 C00079 BC00079
CALL JOB:SEARCH-R1
SET P0311 P0006
SFTON P0311
MOVL C00080 BC00080 V=166.7 PL=0
REFP 3 C00081 BC00081
CALL JOB:SEARCH-R1
SET P0311 P0006
SFTON P0311
MOVL C00082 BC00082 V=166.7 PL=0
SFTOF
'------------------------
'W31.22
'------------------------
MOVL C00083 BC00083 V=500.0
MOVL C00084 BC00084 V=166.7 PL=0
REFP 3 C00085 BC00085
CALL JOB:SEARCH-R1
SET P0312 P0006
SFTON P0312
MOVL C00086 BC00086 V=166.7 PL=0
REFP 3 C00087 BC00087
CALL JOB:SEARCH-R1
SET P0312 P0006
SFTON P0312
MOVL C00088 BC00088 V=166.7 PL=0
SFTOF
'------------------------
'W31.24
'------------------------
MOVL C00089 BC00089 V=500.0
MOVL C00090 BC00090 V=166.7 PL=0
REFP 3 C00091 BC00091
CALL JOB:SEARCH-R1
SET P0313 P0006
SFTON P0313
MOVL C00092 BC00092 V=166.7 PL=0
REFP 3 C00093 BC00093
CALL JOB:SEARCH-R1
SET P0313 P0006
SFTON P0313
MOVL C00094 BC00094 V=166.7 PL=0
SFTOF
'------------------------
'W31.26
'------------------------
MOVL C00095 BC00095 V=500.0
MOVL C00096 BC00096 V=166.7 PL=0
REFP 3 C00097 BC00097
CALL JOB:SEARCH-R1
SET P0314 P0006
SFTON P0314
MOVL C00098 BC00098 V=166.7 PL=0
REFP 3 C00099 BC00099
CALL JOB:SEARCH-R1
SET P0314 P0006
SFTON P0314
MOVL C00100 BC00100 V=166.7 PL=0
SFTOF
'------------------------
MOVL C00101 BC00101 V=333.3
MOVL C00102 BC00102 V=666.7
MOVL C00103 BC00103 V=666.7
MOVL C00104 BC00104 V=666.7
MOVL C00105 BC00105 V=500.0
MOVL C00106 BC00106 V=666.7
MOVL C00107 BC00107 V=666.7
MOVL C00108 BC00108 V=333.3
MOVL C00109 BC00109 V=250.0
'------------------------
'W31.29
'------------------------
MOVL C00110 BC00110 V=166.7 PL=0
REFP 3 C00111 BC00111
CALL JOB:SEARCH-R1
SET P0316 P0006
SFTON P0316
MOVL C00112 BC00112 V=166.7 PL=0
REFP 3 C00113 BC00113
CALL JOB:SEARCH-R1
SET P0316 P0006
SFTON P0316
MOVL C00114 BC00114 V=166.7 PL=0
SFTOF
'------------------------
'W31.31
'------------------------
MOVL C00115 BC00115 V=500.0
MOVL C00116 BC00116 V=166.7 PL=0
REFP 3 C00117 BC00117
CALL JOB:SEARCH-R1
SET P0317 P0006
SFTON P0317
MOVL C00118 BC00118 V=166.7 PL=0
REFP 3 C00119 BC00119
CALL JOB:SEARCH-R1
SET P0317 P0006
SFTON P0317
MOVL C00120 BC00120 V=166.7 PL=0
SFTOF
'------------------------
'W31.32
'------------------------
MOVL C00121 BC00121 V=333.3
MOVL C00122 BC00122 V=333.3
MOVL C00123 BC00123 V=666.7
MOVJ C00124 BC00124 VJ=50.00
MOVJ C00125 BC00125 VJ=50.00
MOVJ C00126 BC00126 VJ=50.00
'W214A P
'------------------------
MOVJ C00127 BC00127 VJ=40.00
MOVL C00128 BC00128 V=166.7 PL=0
REFP 3 C00129 BC00129
CALL JOB:SEARCH-R1
IMOV P0058 V=16.7
SET P0351 P0006
SFTON P0351
REFP 3 C00130 BC00130
CALL JOB:SEARCH-R1
SET P0351 P0006
SFTON P0351
MOVL C00131 BC00131 V=166.7 PL=0
SFTOF
'------------------------
'W219B L
'------------------------
MOVJ C00132 BC00132 VJ=40.00
MOVL C00133 BC00133 V=166.7 PL=0
REFP 3 C00134 BC00134
CALL JOB:SEARCH-R1
IMOV P0058 V=16.7
SET P0352 P0006
SFTON P0352
REFP 3 C00135 BC00135
CALL JOB:SEARCH-R1
SET P0352 P0006
SFTON P0352
MOVL C00136 BC00136 V=166.7 PL=0
SFTOF
'------------------------
'W219B P
'------------------------
MOVJ C00137 BC00137 VJ=40.00
MOVL C00138 BC00138 V=166.7 PL=0
REFP 3 C00139 BC00139
CALL JOB:SEARCH-R1
IMOV P0058 V=16.7
SET P0353 P0006
SFTON P0353
REFP 3 C00140 BC00140
CALL JOB:SEARCH-R1
SET P0353 P0006
SFTON P0353
MOVL C00141 BC00141 V=166.7 PL=0
SFTOF
'------------------------
'W213B L
'------------------------
MOVJ C00142 BC00142 VJ=40.00
MOVL C00143 BC00143 V=166.7 PL=0
REFP 3 C00144 BC00144
CALL JOB:SEARCH-R1
IMOV P0058 V=16.7
SET P0354 P0006
SFTON P0354
REFP 3 C00145 BC00145
CALL JOB:SEARCH-R1
SET P0354 P0006
SFTON P0354
MOVL C00146 BC00146 V=166.7 PL=0
SFTOF
'------------------------
'W213B P
'------------------------
MOVJ C00147 BC00147 VJ=40.00
MOVL C00148 BC00148 V=166.7 PL=0
REFP 3 C00149 BC00149
CALL JOB:SEARCH-R1
IMOV P0058 V=16.7
SET P0355 P0006
SFTON P0355
REFP 3 C00150 BC00150
CALL JOB:SEARCH-R1
SET P0355 P0006
SFTON P0355
MOVL C00151 BC00151 V=166.7 PL=0
SFTOF
'------------------------
'W218B L
'------------------------
MOVJ C00152 BC00152 VJ=40.00
MOVL C00153 BC00153 V=166.7 PL=0
REFP 3 C00154 BC00154
CALL JOB:SEARCH-R1
IMOV P0058 V=16.7
SET P0356 P0006
SFTON P0356
REFP 3 C00155 BC00155
CALL JOB:SEARCH-R1
SET P0356 P0006
SFTON P0356
MOVL C00156 BC00156 V=166.7 PL=0
SFTOF
'------------------------
'W218B P
'------------------------
MOVJ C00157 BC00157 VJ=40.00
MOVL C00158 BC00158 V=166.7 PL=0
REFP 3 C00159 BC00159
CALL JOB:SEARCH-R1
IMOV P0058 V=16.7
SET P0357 P0006
SFTON P0357
REFP 3 C00160 BC00160
CALL JOB:SEARCH-R1
SET P0357 P0006
SFTON P0357
MOVL C00161 BC00161 V=166.7 PL=0
SFTOF
'------------------------
'W215B L
'------------------------
MOVJ C00162 BC00162 VJ=40.00
MOVL C00163 BC00163 V=166.7 PL=0
REFP 3 C00164 BC00164
CALL JOB:SEARCH-R1
IMOV P0058 V=16.7
SET P0358 P0006
SFTON P0358
REFP 3 C00165 BC00165
CALL JOB:SEARCH-R1
SET P0358 P0006
SFTON P0358
MOVL C00166 BC00166 V=166.7 PL=0
SFTOF
'------------------------
'W215B P
'------------------------
MOVL C00167 BC00167 V=666.7
MOVL C00168 BC00168 V=166.7 PL=0
REFP 3 C00169 BC00169
CALL JOB:SEARCH-R1
IMOV P0058 V=16.7
SET P0359 P0006
SFTON P0359
REFP 3 C00170 BC00170
CALL JOB:SEARCH-R1
SET P0359 P0006
SFTON P0359
MOVL C00171 BC00171 V=166.7 PL=0
SFTOF
'------------------------
'W217B L
'------------------------
MOVL C00172 BC00172 V=666.7
MOVL C00173 BC00173 V=166.7 PL=0
REFP 3 C00174 BC00174
CALL JOB:SEARCH-R1
IMOV P0058 V=16.7
SET P0360 P0006
SFTON P0360
REFP 3 C00175 BC00175
CALL JOB:SEARCH-R1
SET P0360 P0006
SFTON P0360
MOVL C00176 BC00176 V=166.7 PL=0
SFTOF
'------------------------
'W217B P
'------------------------
MOVL C00177 BC00177 V=666.7
MOVL C00178 BC00178 V=166.7 PL=0
REFP 3 C00179 BC00179
CALL JOB:SEARCH-R1
IMOV P0058 V=16.7
SET P0361 P0006
SFTON P0361
REFP 3 C00180 BC00180
CALL JOB:SEARCH-R1
SET P0361 P0006
SFTON P0361
MOVL C00181 BC00181 V=166.7 PL=0
SFTOF
MOVL C00182 BC00182 V=333.3
MOVL C00183 BC00183 V=666.7
MOVL C00184 BC00184 V=666.7
MOVJ C00185 BC00185 VJ=50.00
MOVJ C00186 BC00186 VJ=50.00
COMM MOVJ C00187 BC00187 VJ=40.00
COMM MOVJ C00188 BC00188 VJ=40.00
COMM MOVJ C00189 BC00189 VJ=25.00
COMM MOVJ C00190 BC00190 VJ=30.00
COMM MOVJ C00191 BC00191 VJ=30.00
COMM MOVJ C00192 BC00192 VJ=20.00
COMM MOVL C00193 BC00193 V=500.0
COMM '------------------------
COMM 'W27.4
COMM '------------------------
COMM MOVL C00194 BC00194 V=166.7 PL=0
COMM REFP 3 C00195 BC00195
COMM CALL JOB:SEARCH-R1
COMM SET P0401 P0006
COMM SFTON P0401
COMM MOVL C00196 BC00196 V=166.7 PL=0
COMM REFP 3 C00197 BC00197
COMM CALL JOB:SEARCH-R1
COMM SET P0401 P0006
COMM SFTON P0401
COMM MOVL C00198 BC00198 V=166.7 PL=0
COMM SFTOF
COMM '------------------------
COMM 'W27.6
COMM '------------------------
COMM MOVL C00199 BC00199 V=666.7
COMM MOVL C00200 BC00200 V=166.7 PL=0
COMM REFP 3 C00201 BC00201
COMM CALL JOB:SEARCH-R1
COMM SET P0402 P0006
COMM SFTON P0402
COMM MOVL C00202 BC00202 V=166.7 PL=0
COMM REFP 3 C00203 BC00203
COMM CALL JOB:SEARCH-R1
COMM SET P0402 P0006
COMM SFTON P0402
COMM MOVL C00204 BC00204 V=166.7 PL=0
COMM SFTOF
COMM MOVL C00205 BC00205 V=500.0
COMM MOVL C00206 BC00206 V=500.0
COMM '------------------------
COMM 'W27.8
COMM '------------------------
COMM MOVL C00207 BC00207 V=333.3
COMM MOVL C00208 BC00208 V=166.7 PL=0
COMM REFP 3 C00209 BC00209
COMM CALL JOB:SEARCH-R1
COMM SET P0403 P0006
COMM SFTON P0403
COMM MOVL C00210 BC00210 V=166.7 PL=0
COMM REFP 3 C00211 BC00211
COMM CALL JOB:SEARCH-R1
COMM SET P0403 P0006
COMM SFTON P0403
COMM MOVL C00212 BC00212 V=166.7 PL=0
COMM SFTOF
COMM MOVJ C00213 BC00213 VJ=25.00
COMM MOVJ C00214 BC00214 VJ=25.00
COMM MOVJ C00215 BC00215 VJ=30.00
COMM MOVJ C00216 BC00216 VJ=40.00
COMM MOVJ C00217 BC00217 VJ=30.00
COMM '------------------------
COMM 'W27.9
COMM '------------------------
COMM MOVL C00218 BC00218 V=500.0
COMM MOVL C00219 BC00219 V=166.7 PL=0
COMM REFP 3 C00220 BC00220
COMM CALL JOB:SEARCH-R1
COMM SET P0404 P0006
COMM SFTON P0404
COMM MOVL C00221 BC00221 V=166.7 PL=0
COMM REFP 3 C00222 BC00222
COMM CALL JOB:SEARCH-R1
COMM SET P0404 P0006
COMM SFTON P0404
COMM MOVL C00223 BC00223 V=166.7 PL=0
COMM SFTOF
COMM MOVL C00224 BC00224 V=500.0
COMM '------------------------
COMM 'W27.11
COMM '------------------------
COMM MOVL C00225 BC00225 V=500.0
COMM MOVL C00226 BC00226 V=166.7 PL=0
COMM REFP 3 C00227 BC00227
COMM CALL JOB:SEARCH-R1
COMM SET P0405 P0006
COMM SFTON P0405
COMM MOVL C00228 BC00228 V=166.7 PL=0
COMM REFP 3 C00229 BC00229
COMM CALL JOB:SEARCH-R1
COMM SET P0405 P0006
COMM SFTON P0405
COMM MOVL C00230 BC00230 V=166.7 PL=0
COMM SFTOF
COMM MOVL C00231 BC00231 V=666.7
COMM MOVL C00232 BC00232 V=666.7
COMM '------------------------
COMM 'W27.13
COMM '------------------------
COMM MOVL C00233 BC00233 V=333.3
COMM MOVL C00234 BC00234 V=166.7 PL=0
COMM REFP 3 C00235 BC00235
COMM CALL JOB:SEARCH-R1
COMM SET P0406 P0006
COMM SFTON P0406
COMM MOVL C00236 BC00236 V=166.7 PL=0
COMM REFP 3 C00237 BC00237
COMM CALL JOB:SEARCH-R1
COMM SET P0406 P0006
COMM SFTON P0406
COMM MOVL C00238 BC00238 V=166.7 PL=0
COMM SFTOF
COMM '------------------------
COMM 'W27.14
COMM '------------------------
COMM MOVL C00239 BC00239 V=666.7
COMM MOVL C00240 BC00240 V=166.7 PL=0
COMM REFP 3 C00241 BC00241
COMM CALL JOB:SEARCH-R1
COMM SET P0407 P0006
COMM SFTON P0407
COMM MOVL C00242 BC00242 V=166.7 PL=0
COMM REFP 3 C00243 BC00243
COMM CALL JOB:SEARCH-R1
COMM SET P0407 P0006
COMM SFTON P0407
COMM MOVL C00244 BC00244 V=166.7 PL=0
COMM SFTOF
COMM MOVL C00245 BC00245 V=666.7
COMM '------------------------
COMM 'W27.16
COMM '------------------------
COMM MOVL C00246 BC00246 V=333.3
COMM MOVL C00247 BC00247 V=166.7 PL=0
COMM REFP 3 C00248 BC00248
COMM CALL JOB:SEARCH-R1
COMM SET P0408 P0006
COMM SFTON P0408
COMM MOVL C00249 BC00249 V=166.7 PL=0
COMM REFP 3 C00250 BC00250
COMM CALL JOB:SEARCH-R1
COMM SET P0408 P0006
COMM SFTON P0408
COMM MOVL C00251 BC00251 V=166.7 PL=0
COMM SFTOF
COMM MOVL C00252 BC00252 V=666.7
COMM MOVJ C00253 BC00253 VJ=30.00
COMM MOVJ C00254 BC00254 VJ=50.00
COMM MOVJ C00255 BC00255 VJ=40.00
COMM MOVJ C00256 BC00256 VJ=30.00
COMM '------------------------
COMM 'W27.18
COMM '------------------------
COMM MOVL C00257 BC00257 V=333.3
COMM MOVL C00258 BC00258 V=166.7 PL=0
COMM REFP 3 C00259 BC00259
COMM CALL JOB:SEARCH-R1
COMM SET P0409 P0006
COMM SFTON P0409
COMM MOVL C00260 BC00260 V=166.7 PL=0
COMM REFP 3 C00261 BC00261
COMM CALL JOB:SEARCH-R1
COMM SET P0409 P0006
COMM SFTON P0409
COMM MOVL C00262 BC00262 V=166.7 PL=0
COMM SFTOF
COMM '------------------------
COMM 'W27.19
COMM '------------------------
COMM MOVL C00263 BC00263 V=666.7
COMM MOVL C00264 BC00264 V=166.7 PL=0
COMM REFP 3 C00265 BC00265
COMM CALL JOB:SEARCH-R1
COMM SET P0410 P0006
COMM SFTON P0410
COMM MOVL C00266 BC00266 V=166.7 PL=0
COMM REFP 3 C00267 BC00267
COMM CALL JOB:SEARCH-R1
COMM SET P0410 P0006
COMM SFTON P0410
COMM MOVL C00268 BC00268 V=166.7 PL=0
COMM SFTOF
COMM MOVL C00269 BC00269 V=666.7
COMM '------------------------
COMM 'W27.21
COMM '------------------------
COMM MOVL C00270 BC00270 V=166.7 PL=0
COMM REFP 3 C00271 BC00271
COMM CALL JOB:SEARCH-R1
COMM SET P0411 P0006
COMM SFTON P0411
COMM MOVL C00272 BC00272 V=166.7 PL=0
COMM REFP 3 C00273 BC00273
COMM CALL JOB:SEARCH-R1
COMM SET P0411 P0006
COMM SFTON P0411
COMM MOVL C00274 BC00274 V=166.7 PL=0
COMM SFTOF
COMM '------------------------
COMM 'W27.22
COMM '------------------------
COMM MOVL C00275 BC00275 V=666.7
COMM MOVL C00276 BC00276 V=166.7 PL=0
COMM REFP 3 C00277 BC00277
COMM CALL JOB:SEARCH-R1
COMM SET P0412 P0006
COMM SFTON P0412
COMM MOVL C00278 BC00278 V=166.7 PL=0
COMM REFP 3 C00279 BC00279
COMM CALL JOB:SEARCH-R1
COMM SET P0412 P0006
COMM SFTON P0412
COMM MOVL C00280 BC00280 V=166.7 PL=0
COMM SFTOF
COMM MOVL C00281 BC00281 V=666.7
COMM MOVJ C00282 BC00282 VJ=30.00
COMM MOVL C00283 BC00283 V=500.0
COMM '------------------------
COMM 'W27.24
COMM '------------------------
COMM MOVL C00284 BC00284 V=666.7
COMM MOVL C00285 BC00285 V=166.7 PL=0
COMM REFP 3 C00286 BC00286
COMM CALL JOB:SEARCH-R1
COMM SET P0413 P0006
COMM SFTON P0413
COMM MOVL C00287 BC00287 V=166.7 PL=0
COMM REFP 3 C00288 BC00288
COMM CALL JOB:SEARCH-R1
COMM SET P0413 P0006
COMM SFTON P0413
COMM MOVL C00289 BC00289 V=166.7 PL=0
COMM SFTOF
COMM MOVL C00290 BC00290 V=666.7
COMM MOVJ C00291 BC00291 VJ=50.00
COMM MOVJ C00292 BC00292 VJ=50.00
COMM MOVJ C00293 BC00293 VJ=50.00
COMM MOVJ C00294 BC00294 VJ=20.00
COMM MOVJ C00295 BC00295 VJ=10.00
COMM '------------------------
COMM 'W27.26
COMM '------------------------
COMM MOVL C00296 BC00296 V=333.3
COMM MOVL C00297 BC00297 V=166.7 PL=0
COMM REFP 3 C00298 BC00298
COMM CALL JOB:SEARCH-R1
COMM SET P0414 P0006
COMM SFTON P0414
COMM MOVL C00299 BC00299 V=166.7 PL=0
COMM REFP 3 C00300 BC00300
COMM CALL JOB:SEARCH-R1
COMM SET P0414 P0006
COMM SFTON P0414
COMM MOVL C00301 BC00301 V=166.7 PL=0
COMM SFTOF
COMM MOVL C00302 BC00302 V=333.3
COMM MOVJ C00303 BC00303 VJ=30.00
COMM MOVJ C00304 BC00304 VJ=30.00
COMM MOVJ C00305 BC00305 VJ=30.00
COMM GETE D040 P0414 (1)
COMM GETE D041 P0414 (2)
COMM GETE D042 P0414 (3)
COMM SETE P0415 (1) D040
COMM SETE P0415 (2) D041
COMM SETE P0415 (3) D042
COMM '------------------------
COMM 'W27.29
COMM '------------------------
COMM MOVJ C00306 BC00306 VJ=30.00
COMM MOVJ C00307 BC00307 VJ=30.00
COMM MOVL C00308 BC00308 V=333.3
COMM MOVL C00309 BC00309 V=166.7 PL=0
COMM REFP 3 C00310 BC00310
COMM CALL JOB:SEARCH-R1
COMM SET P0416 P0006
COMM SFTON P0416
COMM MOVL C00311 BC00311 V=166.7 PL=0
COMM REFP 3 C00312 BC00312
COMM CALL JOB:SEARCH-R1
COMM SET P0416 P0006
COMM SFTON P0416
COMM MOVL C00313 BC00313 V=166.7 PL=0
COMM SFTOF
COMM '------------------------
COMM 'W27.31
COMM '------------------------
COMM MOVL C00314 BC00314 V=666.7
COMM MOVL C00315 BC00315 V=166.7 PL=0
COMM REFP 3 C00316 BC00316
COMM CALL JOB:SEARCH-R1
COMM SET P0417 P0006
COMM SFTON P0417
COMM MOVL C00317 BC00317 V=166.7 PL=0
COMM REFP 3 C00318 BC00318
COMM CALL JOB:SEARCH-R1
COMM SET P0417 P0006
COMM SFTON P0417
COMM MOVL C00319 BC00319 V=166.7 PL=0
COMM SFTOF
COMM '------------------------
COMM 'W27.32
COMM '------------------------
COMM MOVL C00320 BC00320 V=333.3
MOVJ C00321 BC00321 VJ=50.00
CALL JOB:FRONT_SEARCH_-90ST-1_4690
MOVJ C00322 BC00322 VJ=50.00
MOVJ C00323 BC00323 VJ=50.00
MOVJ C00324 BC00324 VJ=50.00
MOVL C00325 BC00325 V=666.7
MOVJ C00326 BC00326 VJ=30.00
'------------------------
'W31.2
'------------------------
SFTON P0300
MOVL C00327 BC00327 V=333.3
MOVL C00328 BC00328 V=166.7 PL=0
MACRO1 MJ#(0) ARGF10
ARCON
MOVL C00329 BC00329 V=10.8
ARCOF
MOVL C00330 BC00330 V=166.7
SFTOF
'------------------------
'W31.4
'------------------------
SFTON P0301
MOVL C00331 BC00331 V=666.7
MOVL C00332 BC00332 V=166.7 PL=0
ARCON
MOVL C00333 BC00333 V=10.8
ARCOF
MOVL C00334 BC00334 V=166.7
SFTOF
'------------------------
'W31.6
'------------------------
SFTON P0302
MOVL C00335 BC00335 V=666.7
MOVL C00336 BC00336 V=166.7 PL=0
ARCON
MOVL C00337 BC00337 V=10.8
ARCOF
MOVL C00338 BC00338 V=166.7
SFTOF
'------------------------
'W31.8
'------------------------
SFTON P0303
MOVL C00339 BC00339 V=666.7
MOVL C00340 BC00340 V=166.7 PL=0
ARCON
MOVL C00341 BC00341 V=10.8
ARCOF
MOVL C00342 BC00342 V=166.7
SFTOF
'------------------------
'W31.9
'------------------------
SFTON P0304
MOVL C00343 BC00343 V=666.7
MOVL C00344 BC00344 V=166.7 PL=0
ARCON
MOVL C00345 BC00345 V=10.8
ARCOF
MOVL C00346 BC00346 V=166.7
SFTOF
MOVL C00347 BC00347 V=500.0
MOVL C00348 BC00348 V=500.0
MOVJ C00349 BC00349 VJ=50.00
MOVJ C00350 BC00350 VJ=50.00
COMM '::::::::::::::::::::::::::::::::
COMM '::::::::::::::::::::::::::::::::
COMM '::::::::::::::::::::::::::::::::
COMM '::::::::::::::::::::::::::::::::
COMM '::::::::::::::::::::::::::::::::
COMM MOVJ C00351 BC00351 VJ=40.00
COMM MOVJ C00352 BC00352 VJ=40.00
COMM MOVJ C00353 BC00353 VJ=40.00
COMM MOVJ C00354 BC00354 VJ=40.00
COMM MOVJ C00355 BC00355 VJ=40.00
COMM MOVJ C00356 BC00356 VJ=40.00
COMM '------------------------
COMM 'W27.2
COMM '------------------------
COMM MOVL C00357 BC00357 V=500.0
COMM SFTON P0401
COMM MOVL C00358 BC00358 V=166.7 PL=0
COMM MACRO1 MJ#(0) ARGF24
COMM ARCON
COMM MOVL C00359 BC00359 V=7.5
COMM ARCOF
COMM SFTOF
COMM 'BELKA PRZEJAZD
COMM MOVL C00360 BC00360 V=500.0
COMM '------------------------
COMM 'W27.6
COMM '------------------------
COMM SFTON P0402
COMM MOVL C00361 BC00361 V=500.0
COMM MOVL C00362 BC00362 V=166.7 PL=0
COMM MACRO1 MJ#(0) ARGF24
COMM ARCON
COMM MOVL C00363 BC00363 V=7.5
COMM ARCOF
COMM MOVL C00364 BC00364 V=166.7
COMM SFTOF
COMM MOVJ C00365 BC00365 VJ=20.00
COMM '------------------------
COMM 'W27.8
COMM '------------------------
COMM SFTON P0403
COMM MOVL C00366 BC00366 V=500.0
COMM MOVL C00367 BC00367 V=166.7 PL=0
COMM MACRO1 MJ#(0) ARGF24
COMM ARCON
COMM MOVL C00368 BC00368 V=7.5
COMM ARCOF
COMM MOVL C00369 BC00369 V=166.7
COMM SFTOF
COMM MOVL C00370 BC00370 V=500.0
COMM MOVJ C00371 BC00371 VJ=50.00
MOVJ C00372 BC00372 VJ=50.00
MOVJ C00373 BC00373 VJ=50.00
MOVJ C00374 BC00374 VJ=50.00
MOVL C00375 BC00375 V=666.7
'------------------------
'W213A
'------------------------
SFTON P0355
MOVL C00376 BC00376 V=666.7
MOVL C00377 BC00377 V=166.7 PL=0
MACRO1 MJ#(0) ARGF9
ARCON
SFTOF
SFTON P0354
MOVL C00378 BC00378 V=11.2
ARCOF
MOVL C00379 BC00379 V=333.3
SFTOF
MOVJ C00380 BC00380 VJ=50.00
MOVJ C00381 BC00381 VJ=50.00
MOVJ C00382 BC00382 VJ=50.00
MOVJ C00383 BC00383 VJ=50.00
MOVJ C00384 BC00384 VJ=30.00
MOVJ C00385 BC00385 VJ=20.00
MOVJ C00386 BC00386 VJ=20.00
'5.5.1
'------------------------
'W31.11
'------------------------
SFTON P0305
MOVL C00387 BC00387 V=333.3
MOVL C00388 BC00388 V=166.7 PL=0
MACRO1 MJ#(0) ARGF10
ARCON
MOVL C00389 BC00389 V=10.8
ARCOF
MOVL C00390 BC00390 V=166.7
SFTOF
'------------------------
'W31.13
'------------------------
SFTON P0306
MOVL C00391 BC00391 V=500.0
'SPR CZY W DOBRYM MIEJSCU SPOINA
MOVL C00392 BC00392 V=166.7 PL=0
ARCON
MOVL C00393 BC00393 V=10.8
ARCOF
MOVL C00394 BC00394 V=166.7
SFTOF
'------------------------
'W31.14
'------------------------
SFTON P0307
MOVL C00395 BC00395 V=333.3
MOVL C00396 BC00396 V=166.7 PL=0
ARCON
MOVL C00397 BC00397 V=8.3
ARCOF
MOVL C00398 BC00398 V=166.7
SFTOF
MOVL C00399 BC00399 V=333.3
MOVL C00400 BC00400 V=500.0
MOVJ C00401 BC00401 VJ=30.00
MOVJ C00402 BC00402 VJ=30.00
MOVJ C00403 BC00403 VJ=50.00
COMM '::::::::::::::::::::::::::::::::
COMM '::::::::::::::::::::::::::::::::
COMM '------------------------
COMM 'W27.9
COMM '------------------------
COMM '::::::::::::::::::::::::::::::::
COMM '::::::::::::::::::::::::::::::::
COMM MOVJ C00404 BC00404 VJ=25.00
COMM MOVJ C00405 BC00405 VJ=40.00
COMM SFTON P0404
COMM MOVL C00406 BC00406 V=500.0
COMM MOVL C00407 BC00407 V=166.7 PL=0
COMM MACRO1 MJ#(0) ARGF24
COMM ARCON
COMM MOVL C00408 BC00408 V=7.5
COMM ARCOF
COMM MOVL C00409 BC00409 V=166.7
COMM SFTOF
COMM '------------------------
COMM 'W27.11
COMM '------------------------
COMM SFTON P0406
COMM MOVL C00410 BC00410 V=666.7
COMM MOVL C00411 BC00411 V=166.7 PL=0
COMM MACRO1 MJ#(0) ARGF24
COMM ARCON
COMM MOVL C00412 BC00412 V=7.5
COMM ARCOF
COMM MOVL C00413 BC00413 V=166.7
COMM SFTOF
COMM '------------------------
COMM 'W27.13
'------------------------
COMM SFTON P0406
COMM MOVL C00414 BC00414 V=666.7
COMM MOVL C00415 BC00415 V=166.7 PL=0
COMM MACRO1 MJ#(0) ARGF24
COMM ARCON
COMM MOVL C00416 BC00416 V=7.5
COMM ARCOF
COMM MOVL C00417 BC00417 V=166.7
COMM SFTOF
COMM MOVJ C00418 BC00418 VJ=40.00
COMM MOVJ C00419 BC00419 VJ=50.00
COMM MOVJ C00420 BC00420 VJ=50.00
COMM MOVJ C00421 BC00421 VJ=50.00
MOVJ C00422 BC00422 VJ=50.00
'::::::::::::::::::::::::
'::::::::::::::::::::::::
'::::::::::::::::::::::::
'::::::::::::::::::::::::
'::::::::::::::::::::::::
'::::::::::::::::::::::::
'::::::::::::::::::::::::
MOVJ C00423 BC00423 VJ=50.00
MOVJ C00424 BC00424 VJ=50.00
'------------------------
'W214A
'------------------------
SFTON P0351
MOVL C00425 BC00425 V=500.0
MOVL C00426 BC00426 V=166.7 PL=0
MACRO1 MJ#(0) ARGF9
ARCON
MOVL C00427 BC00427 V=11.7
MOVL C00428 BC00428 V=11.0
ARCOF
MOVL C00429 BC00429 V=200.0
SFTOF
MOVJ C00430 BC00430 VJ=50.00
MOVJ C00431 BC00431 VJ=50.00
MOVJ C00432 BC00432 VJ=50.00
MOVJ C00433 BC00433 VJ=40.00
MOVJ C00434 BC00434 VJ=50.00
MOVJ C00435 BC00435 VJ=30.00
MOVJ C00436 BC00436 VJ=30.00
MOVJ C00437 BC00437 VJ=30.00
MOVJ C00438 BC00438 VJ=30.00
'------------------------
'W31.16
'------------------------
SFTON P0308
MOVL C00439 BC00439 V=666.7
MOVL C00440 BC00440 V=166.7 PL=0
MACRO1 MJ#(0) ARGF10
ARCON
MOVL C00441 BC00441 V=10.8
ARCOF
MOVL C00442 BC00442 V=166.7
SFTOF
MOVL C00443 BC00443 V=666.7
MOVL C00444 BC00444 V=666.7
MOVL C00445 BC00445 V=666.7
MOVL C00446 BC00446 V=833.3
MOVL C00447 BC00447 V=666.7
MOVL C00448 BC00448 V=666.7
MOVL C00449 BC00449 V=333.3
MOVL C00450 BC00450 V=333.3
MOVL C00451 BC00451 V=250.0
MOVL C00452 BC00452 V=333.3
'------------------------
'W31.18
'------------------------
SFTON P0309
MOVL C00453 BC00453 V=166.7
MOVL C00454 BC00454 V=83.3 PL=0
ARCON
MOVL C00455 BC00455 V=10.8
ARCOF
MOVL C00456 BC00456 V=166.7
SFTOF
'------------------------
'W31.19
'------------------------
SFTON P0310
MOVL C00457 BC00457 V=333.3
MOVL C00458 BC00458 V=166.7 PL=0
ARCON
MOVL C00459 BC00459 V=10.8
ARCOF
MOVL C00460 BC00460 V=166.7
SFTOF
MOVL C00461 BC00461 V=333.3
MOVL C00462 BC00462 V=500.0
MOVL C00463 BC00463 V=666.7
MOVL C00464 BC00464 V=666.7
MOVJ C00465 BC00465 VJ=40.00
MOVJ C00466 BC00466 VJ=40.00
COMM '::::::::::::::::::::::::
COMM '::::::::::::::::::::::::
COMM '::::::::::::::::::::::::
COMM '::::::::::::::::::::::::
COMM '::::::::::::::::::::::::
COMM '::::::::::::::::::::::::
COMM '::::::::::::::::::::::::
COMM MOVJ C00467 BC00467 VJ=50.00
COMM MOVJ C00468 BC00468 VJ=30.00
COMM '::::::::::::::::::::::::::::::::
COMM '::::::::::::::::::::::::::::::::
COMM '------------------------
COMM 'W27.14
COMM '------------------------
COMM '::::::::::::::::::::::::::::::::
COMM '::::::::::::::::::::::::::::::::
COMM MOVL C00469 BC00469 V=500.0
COMM MOVL C00470 BC00470 V=500.0
COMM SFTON P0407
COMM MOVL C00471 BC00471 V=166.7 PL=0
COMM MACRO1 MJ#(0) ARGF24
COMM ARCON
COMM MOVL C00472 BC00472 V=7.5
COMM ARCOF
COMM MOVL C00473 BC00473 V=166.7
COMM SFTOF
COMM MOVJ C00474 BC00474 VJ=30.00
COMM '------------------------
COMM 'W27.16
COMM '------------------------
COMM SFTON P0408
COMM MOVL C00475 BC00475 V=500.0
COMM MOVL C00476 BC00476 V=166.7 PL=0
COMM MACRO1 MJ#(0) ARGF24
COMM ARCON
COMM MOVL C00477 BC00477 V=6.7
COMM ARCOF
COMM MOVL C00478 BC00478 V=166.7
COMM MOVL C00479 BC00479 V=666.7
COMM MOVJ C00480 BC00480 VJ=50.00
COMM SFTOF
COMM '------------------------
COMM 'W27.18
COMM '------------------------
COMM SFTON P0409
COMM MOVL C00481 BC00481 V=500.0
COMM MOVL C00482 BC00482 V=166.7 PL=0
COMM MACRO1 MJ#(0) ARGF24
COMM ARCON
COMM MOVL C00483 BC00483 V=7.5
COMM ARCOF
COMM MOVL C00484 BC00484 V=166.7
COMM SFTOF
COMM MOVJ C00485 BC00485 VJ=30.00
COMM MOVJ C00486 BC00486 VJ=30.00
COMM MOVJ C00487 BC00487 VJ=40.00
MOVJ C00488 BC00488 VJ=50.00
'::::::::::::::::::::::::
'::::::::::::::::::::::::
'::::::::::::::::::::::::
'::::::::::::::::::::::::
'::::::::::::::::::::::::
'::::::::::::::::::::::::
'::::::::::::::::::::::::
MOVJ C00489 BC00489 VJ=50.00
MOVJ C00490 BC00490 VJ=50.00
'------------------------
'W215A
'------------------------
SFTON P0359
MOVL C00491 BC00491 V=666.7
MOVL C00492 BC00492 V=166.7 PL=0
MACRO1 MJ#(0) ARGF9
ARCON
SFTOF
SFTON P0358
MOVL C00493 BC00493 V=11.7
ARCOF
MOVL C00494 BC00494 V=333.3
SFTOF
MOVJ C00495 BC00495 VJ=50.00
MOVJ C00496 BC00496 VJ=50.00
MOVJ C00497 BC00497 VJ=50.00
MOVJ C00498 BC00498 VJ=50.00
MOVJ C00499 BC00499 VJ=50.00
MOVJ C00500 BC00500 VJ=50.00
MOVJ C00501 BC00501 VJ=50.00
MOVL C00502 BC00502 V=500.0
'------------------------
'W31.21
'------------------------
SFTON P0311
MOVL C00503 BC00503 V=333.3
MOVL C00504 BC00504 V=166.7 PL=0
MACRO1 MJ#(0) ARGF10
ARCON
MOVL C00505 BC00505 V=10.8
ARCOF
MOVL C00506 BC00506 V=166.7
SFTOF
'------------------------
'W31.22
'------------------------
SFTON P0312
MOVL C00507 BC00507 V=666.7
MOVL C00508 BC00508 V=166.7 PL=0
ARCON
MOVL C00509 BC00509 V=10.8
ARCOF
MOVL C00510 BC00510 V=166.7
SFTOF
'------------------------
'W31.24
'------------------------
SFTON P0313
MOVL C00511 BC00511 V=666.7
MOVL C00512 BC00512 V=166.7 PL=0
ARCON
MOVL C00513 BC00513 V=10.8
ARCOF
SFTOF
MOVL C00514 BC00514 V=166.7
MOVL C00515 BC00515 V=166.7
MOVL C00516 BC00516 V=333.3
SFTOF
MOVL C00517 BC00517 V=333.3
MOVJ C00518 BC00518 VJ=30.00
MOVJ C00519 BC00519 VJ=30.00
MOVJ C00520 BC00520 VJ=50.00
MOVJ C00521 BC00521 VJ=50.00
COMM '::::::::::::::::::::::::
COMM '::::::::::::::::::::::::
COMM '::::::::::::::::::::::::
COMM '::::::::::::::::::::::::
COMM '::::::::::::::::::::::::
COMM '::::::::::::::::::::::::
COMM '::::::::::::::::::::::::
COMM MOVJ C00522 BC00522 VJ=50.00
COMM MOVJ C00523 BC00523 VJ=50.00
COMM '::::::::::::::::::::::::::::::::
COMM '::::::::::::::::::::::::::::::::
COMM '------------------------
COMM 'W27.19
COMM '------------------------
COMM '::::::::::::::::::::::::::::::::
COMM '::::::::::::::::::::::::::::::::
COMM MOVJ C00524 BC00524 VJ=30.00
COMM MOVL C00525 BC00525 V=666.7
COMM MOVL C00526 BC00526 V=250.0
COMM SFTON P0410
COMM MOVL C00527 BC00527 V=166.7 PL=0
COMM MACRO1 MJ#(0) ARGF24
COMM ARCON
COMM MOVL C00528 BC00528 V=7.5
COMM ARCOF
COMM MOVL C00529 BC00529 V=166.7
COMM SFTOF
COMM '------------------------
COMM 'W27.21
COMM '------------------------
COMM SFTON P0411
COMM MOVL C00530 BC00530 V=666.7
COMM MOVL C00531 BC00531 V=166.7 PL=0
COMM MACRO1 MJ#(0) ARGF24
COMM ARCON
COMM MOVL C00532 BC00532 V=7.5
COMM ARCOF
COMM MOVL C00533 BC00533 V=250.0
COMM SFTOF
COMM MOVJ C00534 BC00534 VJ=50.00
COMM MOVJ C00535 BC00535 VJ=50.00
COMM MOVJ C00536 BC00536 VJ=50.00
COMM '------------------------
COMM 'W27.22
COMM '------------------------
COMM MOVL C00537 BC00537 V=333.3
COMM MOVL C00538 BC00538 V=333.3
COMM SFTON P0412
COMM MOVL C00539 BC00539 V=166.7 PL=0
COMM MACRO1 MJ#(0) ARGF24
COMM ARCON
COMM MOVL C00540 BC00540 V=7.5
COMM ARCOF
COMM MOVL C00541 BC00541 V=200.0
COMM SFTOF
COMM '::::::::::::::::::::::::
COMM '::::::::::::::::::::::::
COMM '::::::::::::::::::::::::
COMM '::::::::::::::::::::::::
COMM '::::::::::::::::::::::::
COMM '::::::::::::::::::::::::
COMM '::::::::::::::::::::::::
COMM MOVJ C00542 BC00542 VJ=50.00
COMM MOVJ C00543 BC00543 VJ=50.00
COMM MOVJ C00544 BC00544 VJ=50.00
COMM MOVJ C00545 BC00545 VJ=50.00
MOVJ C00546 BC00546 VJ=50.00
'------------------------
'W215A
'------------------------
MOVJ C00547 BC00547 VJ=50.00
MOVJ C00548 BC00548 VJ=50.00
SFTON P0360
MOVL C00549 BC00549 V=500.0
MOVL C00550 BC00550 V=500.0
MOVL C00551 BC00551 V=166.7 PL=0
MACRO1 MJ#(0) ARGF9
ARCON
SFTOF
SFTON P0361
MOVL C00552 BC00552 V=11.7
MOVL C00553 BC00553 V=11.7
ARCOF
MOVL C00554 BC00554 V=500.0
SFTOF
MOVJ C00555 BC00555 VJ=50.00
MOVJ C00556 BC00556 VJ=50.00
MOVJ C00557 BC00557 VJ=50.00
MOVJ C00558 BC00558 VJ=80.00
MOVJ C00559 BC00559 VJ=50.00
MOVJ C00560 BC00560 VJ=50.00
MOVJ C00561 BC00561 VJ=40.00
MOVJ C00562 BC00562 VJ=20.00
MOVL C00563 BC00563 V=333.3
'------------------------
'W31.26
'------------------------
SFTON P0314
MOVL C00564 BC00564 V=833.3
MOVL C00565 BC00565 V=166.7 PL=0
MACRO1 MJ#(0) ARGF10
ARCON
MOVL C00566 BC00566 V=10.8
ARCOF
MOVL C00567 BC00567 V=200.0
SFTOF
'------------------------
MOVL C00568 BC00568 V=500.0
MOVL C00569 BC00569 V=500.0
MOVL C00570 BC00570 V=500.0
MOVL C00571 BC00571 V=500.0
'W31.27
'------------------------
MOVL C00572 BC00572 V=500.0
SFTON P0316
MOVL C00573 BC00573 V=166.7 PL=0
ARCON
MOVL C00574 BC00574 V=10.8
ARCOF
SFTOF
MOVL C00575 BC00575 V=200.0
SFTOF
MOVL C00576 BC00576 V=333.3
MOVL C00577 BC00577 V=416.7
MOVJ C00578 BC00578 VJ=30.00
MOVJ C00579 BC00579 VJ=50.00
MOVJ C00580 BC00580 VJ=50.00
COMM '::::::::::::::::::::::::
COMM '::::::::::::::::::::::::
COMM '::::::::::::::::::::::::
COMM '::::::::::::::::::::::::
COMM '::::::::::::::::::::::::
COMM '::::::::::::::::::::::::
COMM '::::::::::::::::::::::::
COMM MOVJ C00581 BC00581 VJ=50.00
COMM MOVJ C00582 BC00582 VJ=30.00
COMM MOVJ C00583 BC00583 VJ=30.00
COMM MOVJ C00584 BC00584 VJ=40.00
COMM MOVJ C00585 BC00585 VJ=50.00
COMM '::::::::::::::::::::::::::::::::
COMM '::::::::::::::::::::::::::::::::
COMM '------------------------
COMM 'W27.24
COMM '------------------------
COMM '::::::::::::::::::::::::::::::::
COMM '::::::::::::::::::::::::::::::::
COMM SFTON P0413
COMM MOVL C00586 BC00586 V=666.7
COMM MOVL C00587 BC00587 V=500.0
COMM MOVL C00588 BC00588 V=166.7 PL=0
COMM MACRO1 MJ#(0) ARGF24
COMM ARCON
COMM MOVL C00589 BC00589 V=7.5
COMM ARCOF
COMM MOVL C00590 BC00590 V=166.7
COMM SFTOF
COMM MOVJ C00591 BC00591 VJ=30.00
COMM MOVJ C00592 BC00592 VJ=30.00
COMM MOVJ C00593 BC00593 VJ=30.00
COMM '------------------------
COMM 'W27.26
COMM '------------------------
COMM SFTON P0414
COMM MOVL C00594 BC00594 V=333.3
COMM MOVL C00595 BC00595 V=333.3
COMM MOVL C00596 BC00596 V=166.7 PL=0
COMM MACRO1 MJ#(0) ARGF24
COMM ARCON
COMM MOVL C00597 BC00597 V=6.7
COMM ARCOF
COMM MOVL C00598 BC00598 V=200.0
SFTOF
COMM '------------------------
COMM 'W27.27
COMM '------------------------
COMM SFTON P0414
COMM MOVL C00599 BC00599 V=333.3
COMM MOVL C00600 BC00600 V=166.7 PL=0
COMM MACRO1 MJ#(0) ARGF24
COMM ARCON
COMM MOVL C00601 BC00601 V=6.7
COMM ARCOF
COMM MOVL C00602 BC00602 V=200.0
SFTOF
COMM MOVL C00603 BC00603 V=500.0
COMM '::::::::::::::::::::::::
COMM '::::::::::::::::::::::::
COMM '::::::::::::::::::::::::
COMM '::::::::::::::::::::::::
COMM '::::::::::::::::::::::::
COMM '::::::::::::::::::::::::
COMM '::::::::::::::::::::::::
COMM MOVL C00604 BC00604 V=833.3
COMM MOVJ C00605 BC00605 VJ=50.00
COMM MOVJ C00606 BC00606 VJ=50.00
COMM MOVJ C00607 BC00607 VJ=50.00
MOVJ C00608 BC00608 VJ=50.00
'------------------------
'W218A
'------------------------
MOVJ C00609 BC00609 VJ=50.00
MOVJ C00610 BC00610 VJ=50.00
SFTON P0357
MOVL C00611 BC00611 V=500.0
MOVL C00612 BC00612 V=500.0
MOVL C00613 BC00613 V=166.7 PL=0
MACRO1 MJ#(0) ARGF9
ARCON
SFTOF
SFTON P0356
MOVL C00614 BC00614 V=11.7
ARCOF
MOVL C00615 BC00615 V=333.3
SFTOF
MOVJ C00616 BC00616 VJ=50.00
MOVJ C00617 BC00617 VJ=50.00
MOVJ C00618 BC00618 VJ=50.00
MOVJ C00619 BC00619 VJ=50.00
MOVJ C00620 BC00620 VJ=50.00
MOVJ C00621 BC00621 VJ=50.00
MOVL C00622 BC00622 V=500.0
'------------------------
'W31.29
'------------------------
SFTON P0317
MOVL C00623 BC00623 V=333.3
MOVL C00624 BC00624 V=333.3
MOVL C00625 BC00625 V=166.7 PL=0
MOVL C00626 BC00626 V=166.7 PL=0
MACRO1 MJ#(0) ARGF10
ARCON
MOVL C00627 BC00627 V=10.8
ARCOF
MOVL C00628 BC00628 V=166.7
SFTOF
'------------------------
'W31.31
'------------------------
'------------------------
'W31.32
'------------------------
SFTON P0317
MOVL C00629 BC00629 V=166.7 PL=0
ARCON
MOVL C00630 BC00630 V=11.0
ARCOF
SFTOF
MOVL C00631 BC00631 V=333.3
MOVL C00632 BC00632 V=416.7
MOVL C00633 BC00633 V=500.0
MOVL C00634 BC00634 V=500.0
MOVL C00635 BC00635 V=500.0
MOVJ C00636 BC00636 VJ=40.00
MOVJ C00637 BC00637 VJ=50.00
MOVJ C00638 BC00638 VJ=50.00
MOVJ C00639 BC00639 VJ=50.00
COMM '::::::::::::::::::::::::
COMM '::::::::::::::::::::::::
COMM '::::::::::::::::::::::::
COMM '::::::::::::::::::::::::
COMM '::::::::::::::::::::::::
COMM '::::::::::::::::::::::::
COMM '::::::::::::::::::::::::
COMM MOVJ C00640 BC00640 VJ=50.00
COMM MOVJ C00641 BC00641 VJ=50.00
COMM MOVJ C00642 BC00642 VJ=30.00
COMM '::::::::::::::::::::::::::::::::
COMM '::::::::::::::::::::::::::::::::
COMM '------------------------
COMM 'W27.29
COMM '------------------------
COMM '::::::::::::::::::::::::::::::::
COMM '::::::::::::::::::::::::::::::::
COMM SFTON P0416
COMM MOVL C00643 BC00643 V=666.7
COMM MOVL C00644 BC00644 V=166.7 PL=0
COMM MACRO1 MJ#(0) ARGF24
COMM ARCON
COMM MOVL C00645 BC00645 V=6.7
COMM ARCOF
COMM MOVL C00646 BC00646 V=166.7
COMM SFTOF
COMM '------------------------
COMM 'W27.31
COMM '------------------------
COMM SFTON P0417
COMM MOVL C00647 BC00647 V=666.7
COMM MOVL C00648 BC00648 V=166.7
COMM ARCON
COMM MOVL C00649 BC00649 V=7.5
COMM ARCOF
COMM MOVL C00650 BC00650 V=250.0
COMM SFTOF
COMM '------------------------
COMM 'W27.32
COMM '------------------------
COMM '::::::::::::::::::::::::
COMM '::::::::::::::::::::::::
COMM '::::::::::::::::::::::::
COMM '::::::::::::::::::::::::
COMM '::::::::::::::::::::::::
COMM '::::::::::::::::::::::::
COMM '::::::::::::::::::::::::
COMM MOVL C00651 BC00651 V=666.7
COMM MOVJ C00652 BC00652 VJ=40.00
COMM MOVJ C00653 BC00653 VJ=40.00
COMM MOVJ C00654 BC00654 VJ=40.00
COMM MOVJ C00655 BC00655 VJ=40.00
COMM MOVJ C00656 BC00656 VJ=50.00
COMM '------------------------
COMM 'W219A
COMM '------------------------
MOVJ C00657 BC00657 VJ=50.00
MOVJ C00658 BC00658 VJ=50.00
SFTON P0353
MOVL C00659 BC00659 V=666.7
MOVL C00660 BC00660 V=250.0
MOVL C00661 BC00661 V=166.7 PL=0
MACRO1 MJ#(0) ARGF9
ARCON
SFTOF
SFTON P0352
MOVL C00662 BC00662 V=11.7
ARCOF
MOVL C00663 BC00663 V=250.0
SFTOF
MOVJ C00664 BC00664 VJ=50.00
MOVJ C00665 BC00665 VJ=50.00
CALL JOB:FRONT_WELD_-90ST-1_4640
CALL JOB:MOVE_OUT_OF_TUNNEL
END
